LIN {X 0,Y 161.529,Z 676.326,A -85,B 0,C 180,E1 -24059.519,E2 -24059.519} C_VEL
LIN {X 0,Y 165.544,Z 667.107,A -85,B 0,C 180,E1 -24062.772,E2 -24062.772} C_VEL
LIN {X 0,Y 169.219,Z 658.14,A -85,B 0,C 180,E1 -24065.188,E2 -24065.188} C_VEL
LIN {X 0,Y 173.135,Z 647.011,A -85,B 0,C 180,E1 -24067.51,E2 -24067.51} C_VEL
LIN {X 0,Y 176.331,Z 636.142,A -85,B 0,C 180,E1 -24069.252,E2 -24069.252} C_VEL
LIN {X 0,Y 179.205,Z 624.067,A -85,B 0,C 180,E1 -24070.693,E2 -24070.693} C_VEL
LIN {X 0,Y 181.524,Z 611.447,A -85,B 0,C 180,E1 -24071.717,E2 -24071.717} C_VEL
LIN {X 0,Y 182.999,Z 598.442,A -85,B 0,C 180,E1 -24072.415,E2 -24072.415} C_VEL
LIN {X 0,Y 186.753,Z 537.772,A -85,B 0,C 180,E1 -24074.52,E2 -24074.52} C_VEL
LIN {X 0,Y 184.855,Z 513.189,A -85,B 0,C 180,E1 -24076.442,E2 -24076.442} C_VEL
LIN {X 0,Y 184.034,Z 505.216,A -85,B 0,C 180,E1 -24077.157,E2 -24077.157} C_VEL
LIN {X 0,Y 178.957,Z 494.02,A -85,B 0,C 180,E1 -24079.61,E2 -24079.61} C_VEL
LIN {X 0,Y 175.969,Z 487.994,A -85,B 0,C 180,E1 -24081.204,E2 -24081.204} C_VEL
LIN {X 0,Y 173.975,Z 480.034,A -85,B 0,C 180,E1 -24084.963,E2 -24084.963} C_VEL
LIN {X 0,Y 171.968,Z 473.299,A -85,B 0,C 180,E1 -24088.65,E2 -24088.65} C_VEL
LIN {X 0,Y 170.279,Z 468.344,A -85,B 0,C 180,E1 -24091.753,E2 -24091.753} C_VEL
LIN {X 0,Y 168.498,Z 463.406,A -85,B 0,C 180,E1 -24095.348,E2 -24095.348} C_VEL
LIN {X 0,Y 166.157,Z 457.892,A -85,B 0,C 180,E1 -24100.222,E2 -24100.222} C_VEL
LIN {X 0,Y 164.346,Z 453.629,A -85,B 0,C 180,E1 -24105.133,E2 -24105.133} C_VEL
LIN {X 0,Y 162.902,Z 450.174,A -85,B 0,C 180,E1 -24110.063,E2 -24110.063} C_VEL
LIN {X 0,Y 162.272,Z 448.989,A -85,B 0,C 180,E1 -24112.534,E2 -24112.534} C_VEL
LIN {X 0,Y 161.619,Z 446.459,A -85,B 0,C 180,E1 -24120,E2 -24120} C_VEL
LIN {X 0,Y 161.5,Z 446.45,A -85,B 0,C 180,E1 -24122.494,E2 -24122.494} C_VEL
LIN {X 0,Y 161.702,Z 447.367,A -85,B 0,C 180,E1 -24127.492,E2 -24127.492} C_VEL
LIN {X 0,Y 163.472,Z 450.303,A -85,B 0,C 180,E1 -24134.949,E2 -24134.949} C_VEL
LIN {X 0,Y 165.408,Z 453.727,A -85,B 0,C 180,E1 -24139.871,E2 -24139.871} C_VEL
LIN {X 0,Y 166.678,Z 455.735,A -85,B 0,C 180,E1 -24142.302,E2 -24142.302} C_VEL
LIN {X 0,Y 169.717,Z 461.04,A -85,B 0,C 180,E1 -24147.098,E2 -24147.098} C_VEL
LIN {X 0,Y 173.439,Z 467.697,A -85,B 0,C 180,E1 -24151.788,E2 -24151.788} C_VEL
LIN {X 0,Y 177.578,Z 476.226,A -85,B 0,C 180,E1 -24156.417,E2 -24156.417} C_VEL
LIN {X 0,Y 181.019,Z 483.948,A -85,B 0,C 180,E1 -24159.837,E2 -24159.837} C_VEL
LIN {X 0,Y 182.413,Z 487.889,A -85,B 0,C 180,E1 -24161.358,E2 -24161.358} C_VEL
LIN {X 0,Y 183.658,Z 492.595,A -85,B 0,C 180,E1 -24162.176,E2 -24162.176} C_VEL
LIN {X 0,Y 185.304,Z 519.809,A -85,B 0,C 180,E1 -24164.238,E2 -24164.238} C_VEL
LIN {X 0,Y 186.184,Z 541.587,A -85,B 0,C 180,E1 -24165.678,E2 -24165.678} C_VEL
LIN {X 0,Y 182.28,Z 603.538,A -85,B 0,C 180,E1 -24167.839,E2 -24167.839} C_VEL
LIN {X 0,Y 180.62,Z 616.473,A -85,B 0,C 180,E1 -24168.587,E2 -24168.587} C_VEL
LIN {X 0,Y 179.337,Z 623.194,A -85,B 0,C 180,E1 -24169.12,E2 -24169.12} C_VEL
LIN {X 0,Y 177.628,Z 628.814,A -85,B 0,C 180,E1 -24169.52,E2 -24169.52} C_VEL
LIN {X 0,Y 173.272,Z 637.686,A -85,B 0,C 180,E1 -24170.001,E2 -24170.001} C_VEL
LIN {X 0,Y 168.616,Z 646.095,A -85,B 0,C 180,E1 -24170.681,E2 -24170.681} C_VEL
LIN {X 0,Y 166.453,Z 651.018,A -85,B 0,C 180,E1 -24171.432,E2 -24171.432} C_VEL
LIN {X 0,Y 162.264,Z 661.871,A -85,B 0,C 180,E1 -24173.833,E2 -24173.833} C_VEL
LIN {X 0,Y 157.702,Z 672.349,A -85,B 0,C 180,E1 -24176.912,E2 -24176.912} C_VEL
LIN {X 0,Y 154.026,Z 680.047,A -85,B 0,C 180,E1 -24179.873,E2 -24179.873} C_VEL
LIN {X 0,Y 150.219,Z 687.553,A -85,B 0,C 180,E1 -24183.611,E2 -24183.611} C_VEL
LIN {X 0,Y 146.955,Z 693.583,A -85,B 0,C 180,E1 -24187.505,E2 -24187.505} C_VEL
LIN {X 0,Y 144.297,Z 698.343,A -85,B 0,C 180,E1 -24191.543,E2 -24191.543} C_VEL
LIN {X 0,Y 142.495,Z 701.977,A -85,B 0,C 180,E1 -24195.723,E2 -24195.723} C_VEL
LIN {X 0,Y 141.608,Z 703.849,A -85,B 0,C 180,E1 -24198.549,E2 -24198.549} C_VEL
LIN {X 0,Y 141.003,Z 705.258,A -85,B 0,C 180,E1 -24201.4,E2 -24201.4} C_VEL
LIN {X 0,Y 140.695,Z 706.254,A -85,B 0,C 180,E1 -24204.266,E2 -24204.266} C_VEL
LIN {X 0,Y 140.569,Z 707.048,A -85,B 0,C 180,E1 -24209.356,E2 -24209.356} C_VEL
LIN {X 0,Y 140.551,Z 706.847,A -85,B 0,C 180,E1 -24212.866,E2 -24212.866} C_VEL
LIN {X 0,Y 140.695,Z 706.23,A -85,B 0,C 180,E1 -24215.733,E2 -24215.733} C_VEL
LIN {X 0,Y 141.003,Z 705.224,A -85,B 0,C 180,E1 -24218.599,E2 -24218.599} C_VEL
LIN {X 0,Y 141.609,Z 703.795,A -85,B 0,C 180,E1 -24221.45,E2 -24221.45} C_VEL
LIN {X 0,Y 143.026,Z 700.831,A -85,B 0,C 180,E1 -24225.679,E2 -24225.679} C_VEL
LIN {X 0,Y 145.08,Z 696.809,A -85,B 0,C 180,E1 -24229.821,E2 -24229.821} C_VEL
LIN {X 0,Y 148.537,Z 690.612,A -85,B 0,C 180,E1 -24234.456,E2 -24234.456} C_VEL
LIN {X 0,Y 152.052,Z 684.024,A -85,B 0,C 180,E1 -24238.172,E2 -24238.172} C_VEL
LIN {X 0,Y 155.429,Z 676.931,A -85,B 0,C 180,E1 -24241.332,E2 -24241.332} C_VEL
LIN {X 0,Y 159.305,Z 668.576,A -85,B 0,C 180,E1 -24244.228,E2 -24244.228} C_VEL
LIN {X 0,Y 163.571,Z 658.245,A -85,B 0,C 180,E1 -24246.979,E2 -24246.979} C_VEL
LIN {X 0,Y 167.746,Z 646.617,A -85,B 0,C 180,E1 -24249.322,E2 -24249.322} C_VEL
LIN {X 0,Y 169.092,Z 643.157,A -85,B 0,C 180,E1 -24249.913,E2 -24249.913} C_VEL
LIN {X 0,Y 176.202,Z 640.592,A -85,B 0,C 180,E1 -24252.692,E2 -24252.692} C_VEL
LIN {X 0,Y 186.438,Z 636.605,A -85,B 0,C 180,E1 -24255.744,E2 -24255.744} C_VEL
LIN {X 0,Y 197.602,Z 631.417,A -85,B 0,C 180,E1 -24258.322,E2 -24258.322} C_VEL
LIN {X 0,Y 199.719,Z 630.307,A -85,B 0,C 180,E1 -24258.745,E2 -24258.745} C_VEL
LIN {X 0,Y 200.899,Z 629.352,A -85,B 0,C 180,E1 -24259.557,E2 -24259.557} C_VEL
LIN {X 0,Y 192.906,Z 631.179,A -85,B 0,C 180,E1 -24261.731,E2 -24261.731} C_VEL
LIN {X 0,Y 183.116,Z 632.283,A -85,B 0,C 180,E1 -24264.851,E2 -24264.851} C_VEL
LIN {X 0,Y 174.085,Z 632.009,A -85,B 0,C 180,E1 -24268.344,E2 -24268.344} C_VEL
LIN {X 0,Y 166.006,Z 630.276,A -85,B 0,C 180,E1 -24272.245,E2 -24272.245} C_VEL
LIN {X 0,Y 158.996,Z 627.135,A -85,B 0,C 180,E1 -24276.558,E2 -24276.558} C_VEL
LIN {X 0,Y 153.197,Z 622.556,A -85,B 0,C 180,E1 -24281.269,E2 -24281.269} C_VEL
LIN {X 0,Y 148.739,Z 616.364,A -85,B 0,C 180,E1 -24286.335,E2 -24286.335} C_VEL
LIN {X 0,Y 146.114,Z 609.561,A -85,B 0,C 180,E1 -24291.007,E2 -24291.007} C_VEL
LIN {X 0,Y 144.181,Z 601.237,A -85,B 0,C 180,E1 -24295.807,E2 -24295.807} C_VEL
LIN {X 0,Y 143.45,Z 590.998,A -85,B 0,C 180,E1 -24300.702,E2 -24300.702} C_VEL
LIN {X 0,Y 143.461,Z 580.348,A -85,B 0,C 180,E1 -24304.918,E2 -24304.918} C_VEL
LIN {X 0,Y 143.996,Z 568.578,A -85,B 0,C 180,E1 -24308.773,E2 -24308.773} C_VEL
LIN {X 0,Y 144.72,Z 555.919,A -85,B 0,C 180,E1 -24312.081,E2 -24312.081} C_VEL
LIN {X 0,Y 145.46,Z 543.621,A -85,B 0,C 180,E1 -24314.694,E2 -24314.694} C_VEL
LIN {X 0,Y 146.296,Z 529.161,A -85,B 0,C 180,E1 -24317.112,E2 -24317.112} C_VEL
LIN {X 0,Y 146.975,Z 515.38,A -85,B 0,C 180,E1 -24318.831,E2 -24318.831} C_VEL
LIN {X 0,Y 147.665,Z 492.766,A -85,B 0,C 180,E1 -24321.096,E2 -24321.096} C_VEL
LIN {X 0,Y 147.855,Z 488.31,A -85,B 0,C 180,E1 -24321.891,E2 -24321.891} C_VEL
LIN {X 0,Y 148.091,Z 487.68,A -85,B 0,C 180,E1 -24322.313,E2 -24322.313} C_VEL
LIN {X 0,Y 149.825,Z 486.897,A -85,B 0,C 180,E1 -24323.498,E2 -24323.498} C_VEL
LIN {X 0,Y 152.829,Z 484.252,A -85,B 0,C 180,E1 -24324.449,E2 -24324.449} C_VEL
LIN {X 0,Y 154.839,Z 483.406,A -85,B 0,C 180,E1 -24325.545,E2 -24325.545} C_VEL
LIN {X 0,Y 160.173,Z 479.672,A -85,B 0,C 180,E1 -24327.434,E2 -24327.434} C_VEL
LIN {X 0,Y 162.59,Z 478.361,A -85,B 0,C 180,E1 -24328.391,E2 -24328.391} C_VEL
LIN {X 0,Y 165.368,Z 476.481,A -85,B 0,C 180,E1 -24329.258,E2 -24329.258} C_VEL
LIN {X 0,Y 166.775,Z 477.154,A -85,B 0,C 180,E1 -24330.377,E2 -24330.377} C_VEL
LIN {X 0,Y 168.809,Z 483.952,A -85,B 0,C 180,E1 -24334.196,E2 -24334.196} C_VEL
LIN {X 0,Y 169.895,Z 488.503,A -85,B 0,C 180,E1 -24336.503,E2 -24336.503} C_VEL
LIN {X 0,Y 174.656,Z 497.876,A -85,B 0,C 180,E1 -24339.176,E2 -24339.176} C_VEL
LIN {X 0,Y 178.713,Z 507.05,A -85,B 0,C 180,E1 -24341.295,E2 -24341.295} C_VEL
LIN {X 0,Y 179.393,Z 509.152,A -85,B 0,C 180,E1 -24341.666,E2 -24341.666} C_VEL
LIN {X 0,Y 181.143,Z 532.748,A -85,B 0,C 180,E1 -24343.63,E2 -24343.63} C_VEL
LIN {X 0,Y 181.538,Z 539.6,A -85,B 0,C 180,E1 -24344.143,E2 -24344.143} C_VEL
LIN {X 0,Y 177.35,Z 602.381,A -85,B 0,C 180,E1 -24346.383,E2 -24346.383} C_VEL
LIN {X 0,Y 175.415,Z 615.477,A -85,B 0,C 180,E1 -24347.168,E2 -24347.168} C_VEL
LIN {X 0,Y 172.761,Z 628.498,A -85,B 0,C 180,E1 -24348.425,E2 -24348.425} C_VEL
LIN {X 0,Y 169.587,Z 640.39,A -85,B 0,C 180,E1 -24350.033,E2 -24350.033} C_VEL
LIN {X 0,Y 165.778,Z 651.672,A -85,B 0,C 180,E1 -24352.069,E2 -24352.069} C_VEL
LIN {X 0,Y 161.788,Z 661.855,A -85,B 0,C 180,E1 -24354.479,E2 -24354.479} C_VEL
LIN {X 0,Y 158.169,Z 670.201,A -85,B 0,C 180,E1 -24357.023,E2 -24357.023} C_VEL
LIN {X 0,Y 154.607,Z 677.898,A -85,B 0,C 180,E1 -24359.998,E2 -24359.998} C_VEL
LIN {X 0,Y 150.701,Z 685.393,A -85,B 0,C 180,E1 -24363.702,E2 -24363.702} C_VEL
LIN {X 0,Y 147.336,Z 691.406,A -85,B 0,C 180,E1 -24367.567,E2 -24367.567} C_VEL
LIN {X 0,Y 144.701,Z 696.159,A -85,B 0,C 180,E1 -24371.597,E2 -24371.597} C_VEL
LIN {X 0,Y 142.761,Z 699.794,A -85,B 0,C 180,E1 -24375.751,E2 -24375.751} C_VEL
LIN {X 0,Y 141.822,Z 701.664,A -85,B 0,C 180,E1 -24378.567,E2 -24378.567} C_VEL
LIN {X 0,Y 141.13,Z 703.088,A -85,B 0,C 180,E1 -24381.409,E2 -24381.409} C_VEL
LIN {X 0,Y 140.727,Z 704.087,A -85,B 0,C 180,E1 -24384.268,E2 -24384.268} C_VEL
LIN {X 0,Y 140.538,Z 704.701,A -85,B 0,C 180,E1 -24387.134,E2 -24387.134} C_VEL
LIN {X 0,Y 140.528,Z 704.932,A -85,B 0,C 180,E1 -24390,E2 -24390} C_VEL
LIN {X 0,Y 140.538,Z 704.731,A -85,B 0,C 180,E1 -24392.867,E2 -24392.867} C_VEL
LIN {X 0,Y 140.71,Z 704.137,A -85,B 0,C 180,E1 -24395.733,E2 -24395.733} C_VEL
LIN {X 0,Y 141.083,Z 703.158,A -85,B 0,C 180,E1 -24398.595,E2 -24398.595} C_VEL
LIN {X 0,Y 141.74,Z 701.773,A -85,B 0,C 180,E1 -24401.44,E2 -24401.44} C_VEL
LIN {X 0,Y 143.28,Z 698.869,A -85,B 0,C 180,E1 -24405.652,E2 -24405.652} C_VEL
LIN {X 0,Y 145.379,Z 694.923,A -85,B 0,C 180,E1 -24409.78,E2 -24409.78} C_VEL
LIN {X 0,Y 148.322,Z 689.807,A -85,B 0,C 180,E1 -24413.751,E2 -24413.751} C_VEL
LIN {X 0,Y 151.813,Z 683.36,A -85,B 0,C 180,E1 -24417.577,E2 -24417.577} C_VEL
LIN {X 0,Y 155.861,Z 675.352,A -85,B 0,C 180,E1 -24421.234,E2 -24421.234} C_VEL
LIN {X 0,Y 159.596,Z 667.153,A -85,B 0,C 180,E1 -24424.158,E2 -24424.158} C_VEL
LIN {X 0,Y 163.938,Z 657.038,A -85,B 0,C 180,E1 -24426.883,E2 -24426.883} C_VEL
LIN {X 0,Y 168.049,Z 645.661,A -85,B 0,C 180,E1 -24429.239,E2 -24429.239} C_VEL
LIN {X 0,Y 171.384,Z 634.406,A -85,B 0,C 180,E1 -24431.005,E2 -24431.005} C_VEL
LIN {X 0,Y 174.427,Z 621.607,A -85,B 0,C 180,E1 -24432.446,E2 -24432.446} C_VEL
LIN {X 0,Y 176.664,Z 609.011,A -85,B 0,C 180,E1 -24433.416,E2 -24433.416} C_VEL
LIN {X 0,Y 178.074,Z 595.759,A -85,B 0,C 180,E1 -24434.041,E2 -24434.041} C_VEL
LIN {X 0,Y 181.707,Z 538.828,A -85,B 0,C 180,E1 -24436.043,E2 -24436.043} C_VEL
LIN {X 0,Y 180.027,Z 514.977,A -85,B 0,C 180,E1 -24437.973,E2 -24437.973} C_VEL
LIN {X 0,Y 179.352,Z 508.348,A -85,B 0,C 180,E1 -24438.604,E2 -24438.604} C_VEL
LIN {X 0,Y 174.464,Z 497.305,A -85,B 0,C 180,E1 -24441.159,E2 -24441.159} C_VEL
LIN {X 0,Y 169.725,Z 487.967,A -85,B 0,C 180,E1 -24443.908,E2 -24443.908} C_VEL
LIN {X 0,Y 167.852,Z 480.601,A -85,B 0,C 180,E1 -24447.79,E2 -24447.79} C_VEL
LIN {X 0,Y 166.296,Z 475.411,A -85,B 0,C 180,E1 -24450.921,E2 -24450.921} C_VEL
LIN {X 0,Y 164.426,Z 470.181,A -85,B 0,C 180,E1 -24454.695,E2 -24454.695} C_VEL
LIN {X 0,Y 162.79,Z 465.679,A -85,B 0,C 180,E1 -24458.471,E2 -24458.471} C_VEL
LIN {X 0,Y 161.257,Z 461.982,A -85,B 0,C 180,E1 -24462.237,E2 -24462.237} C_VEL
LIN {X 0,Y 159.754,Z 458.091,A -85,B 0,C 180,E1 -24467.293,E2 -24467.293} C_VEL
LIN {X 0,Y 159.225,Z 456.473,A -85,B 0,C 180,E1 -24469.831,E2 -24469.831} C_VEL
LIN {X 0,Y 158.634,Z 455.181,A -85,B 0,C 180,E1 -24472.362,E2 -24472.362} C_VEL
LIN {X 0,Y 157.973,Z 452.588,A -85,B 0,C 180,E1 -24480,E2 -24480} C_VEL
LIN {X 0,Y 157.969,Z 452.641,A -85,B 0,C 180,E1 -24482.55,E2 -24482.55} C_VEL
LIN {X 0,Y 158.328,Z 453.67,A -85,B 0,C 180,E1 -24487.653,E2 -24487.653} C_VEL
LIN {X 0,Y 160.107,Z 456.758,A -85,B 0,C 180,E1 -24495.27,E2 -24495.27} C_VEL
LIN {X 0,Y 162.611,Z 461.061,A -85,B 0,C 180,E1 -24501.312,E2 -24501.312} C_VEL
LIN {X 0,Y 165.743,Z 466.703,A -85,B 0,C 180,E1 -24506.574,E2 -24506.574} C_VEL
LIN {X 0,Y 168.843,Z 472.526,A -85,B 0,C 180,E1 -24510.816,E2 -24510.816} C_VEL
LIN {X 0,Y 172.221,Z 479.503,A -85,B 0,C 180,E1 -24514.842,E2 -24514.842} C_VEL
LIN {X 0,Y 175.924,Z 488.125,A -85,B 0,C 180,E1 -24518.953,E2 -24518.953} C_VEL
LIN {X 0,Y 178.149,Z 492.16,A -85,B 0,C 180,E1 -24520.148,E2 -24520.148} C_VEL
LIN {X 0,Y 178.999,Z 495.228,A -85,B 0,C 180,E1 -24520.656,E2 -24520.656} C_VEL
LIN {X 0,Y 180.507,Z 523.357,A -85,B 0,C 180,E1 -24522.85,E2 -24522.85} C_VEL
LIN {X 0,Y 181.158,Z 542.035,A -85,B 0,C 180,E1 -24524.124,E2 -24524.124} C_VEL
LIN {X 0,Y 177.056,Z 603.874,A -85,B 0,C 180,E1 -24526.309,E2 -24526.309} C_VEL
LIN {X 0,Y 175.358,Z 616.466,A -85,B 0,C 180,E1 -24527.052,E2 -24527.052} C_VEL
LIN {X 0,Y 172.683,Z 629.321,A -85,B 0,C 180,E1 -24528.206,E2 -24528.206} C_VEL
LIN {X 0,Y 169.696,Z 640.745,A -85,B 0,C 180,E1 -24529.675,E2 -24529.675} C_VEL
LIN {X 0,Y 166.453,Z 651.018,A -85,B 0,C 180,E1 -24531.432,E2 -24531.432} C_VEL
LIN {X 0,Y 164.182,Z 655.911,A -85,B 0,C 180,E1 -24532.271,E2 -24532.271} C_VEL
LIN {X 0,Y 158.789,Z 663.497,A -85,B 0,C 180,E1 -24533.492,E2 -24533.492} C_VEL
LIN {X 0,Y 153.178,Z 670.57,A -85,B 0,C 180,E1 -24535.004,E2 -24535.004} C_VEL
LIN {X 0,Y 150.621,Z 674.63,A -85,B 0,C 180,E1 -24536.298,E2 -24536.298} C_VEL
LIN {X 0,Y 146.746,Z 682.242,A -85,B 0,C 180,E1 -24539.549,E2 -24539.549} C_VEL
LIN {X 0,Y 143.238,Z 688.611,A -85,B 0,C 180,E1 -24543.008,E2 -24543.008} C_VEL
LIN {X 0,Y 140.417,Z 693.532,A -85,B 0,C 180,E1 -24546.396,E2 -24546.396} C_VEL
LIN {X 0,Y 137.559,Z 698.291,A -85,B 0,C 180,E1 -24550.604,E2 -24550.604} C_VEL
LIN {X 0,Y 135.585,Z 701.924,A -85,B 0,C 180,E1 -24554.979,E2 -24554.979} C_VEL
LIN {X 0,Y 134.626,Z 703.796,A -85,B 0,C 180,E1 -24557.947,E2 -24557.947} C_VEL
LIN {X 0,Y 133.976,Z 705.205,A -85,B 0,C 180,E1 -24560.945,E2 -24560.945} C_VEL
LIN {X 0,Y 133.631,Z 706.201,A -85,B 0,C 180,E1 -24563.962,E2 -24563.962} C_VEL
LIN {X 0,Y 133.471,Z 706.808,A -85,B 0,C 180,E1 -24566.981,E2 -24566.981} C_VEL
LIN {X 0,Y 133.499,Z 707.02,A -85,B 0,C 180,E1 -24570,E2 -24570} C_VEL
LIN {X 0,Y 133.47,Z 706.793,A -85,B 0,C 180,E1 -24573.018,E2 -24573.018} C_VEL
LIN {X 0,Y 133.63,Z 706.175,A -85,B 0,C 180,E1 -24576.037,E2 -24576.037} C_VEL
LIN {X 0,Y 133.976,Z 705.169,A -85,B 0,C 180,E1 -24579.054,E2 -24579.054} C_VEL
LIN {X 0,Y 134.627,Z 703.74,A -85,B 0,C 180,E1 -24582.052,E2 -24582.052} C_VEL
LIN {X 0,Y 136.174,Z 700.776,A -85,B 0,C 180,E1 -24586.49,E2 -24586.49} C_VEL
LIN {X 0,Y 138.412,Z 696.755,A -85,B 0,C 180,E1 -24590.82,E2 -24590.82} C_VEL
LIN {X 0,Y 142.07,Z 690.558,A -85,B 0,C 180,E1 -24595.648,E2 -24595.648} C_VEL
LIN {X 0,Y 146.049,Z 683.455,A -85,B 0,C 180,E1 -24599.776,E2 -24599.776} C_VEL
LIN {X 0,Y 150.164,Z 675.323,A -85,B 0,C 180,E1 -24603.362,E2 -24603.362} C_VEL
LIN {X 0,Y 154.361,Z 666.605,A -85,B 0,C 180,E1 -24606.291,E2 -24606.291} C_VEL
LIN {X 0,Y 158.907,Z 655.881,A -85,B 0,C 180,E1 -24609.067,E2 -24609.067} C_VEL
LIN {X 0,Y 162.858,Z 645.067,A -85,B 0,C 180,E1 -24611.155,E2 -24611.155} C_VEL
LIN {X 0,Y 164.166,Z 642.142,A -85,B 0,C 180,E1 -24611.674,E2 -24611.674} C_VEL
LIN {X 0,Y 171.063,Z 640.15,A -85,B 0,C 180,E1 -24614.301,E2 -24614.301} C_VEL
LIN {X 0,Y 181.547,Z 636.713,A -85,B 0,C 180,E1 -24617.351,E2 -24617.351} C_VEL
LIN {X 0,Y 190.232,Z 633.287,A -85,B 0,C 180,E1 -24619.357,E2 -24619.357} C_VEL
LIN {X 0,Y 189.199,Z 633.24,A -85,B 0,C 180,E1 -24620.008,E2 -24620.008} C_VEL
LIN {X 0,Y 182.475,Z 633.879,A -85,B 0,C 180,E1 -24621.958,E2 -24621.958} C_VEL
LIN {X 0,Y 172.7,Z 633.752,A -85,B 0,C 180,E1 -24625.269,E2 -24625.269} C_VEL
LIN {X 0,Y 163.858,Z 632.238,A -85,B 0,C 180,E1 -24629.023,E2 -24629.023} C_VEL
LIN {X 0,Y 156,Z 629.292,A -85,B 0,C 180,E1 -24633.223,E2 -24633.223} C_VEL
LIN {X 0,Y 149.33,Z 624.929,A -85,B 0,C 180,E1 -24637.882,E2 -24637.882} C_VEL
LIN {X 0,Y 143.999,Z 619.088,A -85,B 0,C 180,E1 -24642.972,E2 -24642.972} C_VEL
LIN {X 0,Y 140.286,Z 611.576,A -85,B 0,C 180,E1 -24648.44,E2 -24648.44} C_VEL
LIN {X 0,Y 137.94,Z 603.393,A -85,B 0,C 180,E1 -24653.417,E2 -24653.417} C_VEL
LIN {X 0,Y 136.694,Z 593.477,A -85,B 0,C 180,E1 -24658.527,E2 -24658.527} C_VEL
LIN {X 0,Y 136.479,Z 583.189,A -85,B 0,C 180,E1 -24662.952,E2 -24662.952} C_VEL
LIN {X 0,Y 136.852,Z 571.757,A -85,B 0,C 180,E1 -24667.006,E2 -24667.006} C_VEL
LIN {X 0,Y 137.419,Z 560.623,A -85,B 0,C 180,E1 -24670.312,E2 -24670.312} C_VEL
LIN {X 0,Y 138.073,Z 549.186,A -85,B 0,C 180,E1 -24673.08,E2 -24673.08} C_VEL
LIN {X 0,Y 138.971,Z 533.049,A -85,B 0,C 180,E1 -24676.176,E2 -24676.176} C_VEL
LIN {X 0,Y 139.44,Z 524.996,A -85,B 0,C 180,E1 -24677.792,E2 -24677.792} C_VEL
LIN {X 0,Y 139.758,Z 522.696,A -85,B 0,C 180,E1 -24678.603,E2 -24678.603} C_VEL
LIN {X 0,Y 140.364,Z 521.75,A -85,B 0,C 180,E1 -24679.373,E2 -24679.373} C_VEL
LIN {X 0,Y 141.679,Z 518.777,A -85,B 0,C 180,E1 -24680.413,E2 -24680.413} C_VEL
LIN {X 0,Y 143.518,Z 513.065,A -85,B 0,C 180,E1 -24681.549,E2 -24681.549} C_VEL
LIN {X 0,Y 147.072,Z 499.47,A -85,B 0,C 180,E1 -24683.219,E2 -24683.219} C_VEL
LIN {X 0,Y 148.576,Z 493.924,A -85,B 0,C 180,E1 -24683.893,E2 -24683.893} C_VEL
LIN {X 0,Y 150.073,Z 492.752,A -85,B 0,C 180,E1 -24685.02,E2 -24685.02} C_VEL
LIN {X 0,Y 152.013,Z 489.85,A -85,B 0,C 180,E1 -24686.238,E2 -24686.238} C_VEL
LIN {X 0,Y 153.569,Z 488.674,A -85,B 0,C 180,E1 -24687.235,E2 -24687.235} C_VEL
LIN {X 0,Y 158.932,Z 484.913,A -85,B 0,C 180,E1 -24689.106,E2 -24689.106} C_VEL
LIN {X 0,Y 161.439,Z 483.58,A -85,B 0,C 180,E1 -24690.042,E2 -24690.042} C_VEL
LIN {X 0,Y 162.751,Z 484.509,A -85,B 0,C 180,E1 -24691.211,E2 -24691.211} C_VEL
LIN {X 0,Y 163.667,Z 488.248,A -85,B 0,C 180,E1 -24693.403,E2 -24693.403} C_VEL
LIN {X 0,Y 167.785,Z 496.259,A -85,B 0,C 180,E1 -24696.091,E2 -24696.091} C_VEL
LIN {X 0,Y 171.493,Z 503.922,A -85,B 0,C 180,E1 -24698.265,E2 -24698.265} C_VEL
LIN {X 0,Y 174.778,Z 511.715,A -85,B 0,C 180,E1 -24700.099,E2 -24700.099} C_VEL
LIN {X 0,Y 176.255,Z 533.448,A -85,B 0,C 180,E1 -24701.98,E2 -24701.98} C_VEL
LIN {X 0,Y 176.616,Z 539.816,A -85,B 0,C 180,E1 -24702.488,E2 -24702.488} C_VEL
LIN {X 0,Y 172.26,Z 602.734,A -85,B 0,C 180,E1 -24704.775,E2 -24704.775} C_VEL
LIN {X 0,Y 170.296,Z 615.503,A -85,B 0,C 180,E1 -24705.55,E2 -24705.55} C_VEL
LIN {X 0,Y 167.521,Z 628.535,A -85,B 0,C 180,E1 -24706.815,E2 -24706.815} C_VEL
LIN {X 0,Y 164.215,Z 640.434,A -85,B 0,C 180,E1 -24708.443,E2 -24708.443} C_VEL
LIN {X 0,Y 160.249,Z 651.719,A -85,B 0,C 180,E1 -24710.512,E2 -24710.512} C_VEL
LIN {X 0,Y 156.073,Z 661.904,A -85,B 0,C 180,E1 -24712.967,E2 -24712.967} C_VEL
LIN {X 0,Y 152.238,Z 670.253,A -85,B 0,C 180,E1 -24715.562,E2 -24715.562} C_VEL
LIN {X 0,Y 147.773,Z 679.293,A -85,B 0,C 180,E1 -24719.252,E2 -24719.252} C_VEL
LIN {X 0,Y 143.745,Z 686.544,A -85,B 0,C 180,E1 -24723.112,E2 -24723.112} C_VEL
LIN {X 0,Y 139.751,Z 693.19,A -85,B 0,C 180,E1 -24727.842,E2 -24727.842} C_VEL
LIN {X 0,Y 137.215,Z 697.553,A -85,B 0,C 180,E1 -24732.103,E2 -24732.103} C_VEL
LIN {X 0,Y 135.874,Z 699.848,A -85,B 0,C 180,E1 -24735.012,E2 -24735.012} C_VEL
LIN {X 0,Y 134.85,Z 701.719,A -85,B 0,C 180,E1 -24737.968,E2 -24737.968} C_VEL
LIN {X 0,Y 134.108,Z 703.143,A -85,B 0,C 180,E1 -24740.955,E2 -24740.955} C_VEL
LIN {X 0,Y 133.466,Z 704.755,A -85,B 0,C 180,E1 -24746.982,E2 -24746.982} C_VEL
LIN {X 0,Y 133.45,Z 704.986,A -85,B 0,C 180,E1 -24750,E2 -24750} C_VEL
LIN {X 0,Y 133.465,Z 704.785,A -85,B 0,C 180,E1 -24753.019,E2 -24753.019} C_VEL
LIN {X 0,Y 133.645,Z 704.19,A -85,B 0,C 180,E1 -24756.038,E2 -24756.038} C_VEL
LIN {X 0,Y 134.068,Z 703.211,A -85,B 0,C 180,E1 -24759.049,E2 -24759.049} C_VEL
LIN {X 0,Y 134.779,Z 701.826,A -85,B 0,C 180,E1 -24762.04,E2 -24762.04} C_VEL
LIN {X 0,Y 136.437,Z 698.922,A -85,B 0,C 180,E1 -24766.458,E2 -24766.458} C_VEL
LIN {X 0,Y 138.697,Z 694.975,A -85,B 0,C 180,E1 -24770.776,E2 -24770.776} C_VEL
LIN {X 0,Y 141.843,Z 689.857,A -85,B 0,C 180,E1 -24774.908,E2 -24774.908} C_VEL
LIN {X 0,Y 145.552,Z 683.41,A -85,B 0,C 180,E1 -24778.873,E2 -24778.873} C_VEL
LIN {X 0,Y 149.672,Z 675.688,A -85,B 0,C 180,E1 -24782.524,E2 -24782.524} C_VEL
LIN {X 0,Y 153.77,Z 667.198,A -85,B 0,C 180,E1 -24785.644,E2 -24785.644} C_VEL
LIN {X 0,Y 157.819,Z 658.223,A -85,B 0,C 180,E1 -24788.162,E2 -24788.162} C_VEL
LIN {X 0,Y 162.114,Z 647.086,A -85,B 0,C 180,E1 -24790.564,E2 -24790.564} C_VEL
LIN {X 0,Y 165.596,Z 636.203,A -85,B 0,C 180,E1 -24792.358,E2 -24792.358} C_VEL
LIN {X 0,Y 168.71,Z 624.102,A -85,B 0,C 180,E1 -24793.833,E2 -24793.833} C_VEL
LIN {X 0,Y 171.303,Z 610.821,A -85,B 0,C 180,E1 -24794.918,E2 -24794.918} C_VEL
LIN {X 0,Y 172.837,Z 597.976,A -85,B 0,C 180,E1 -24795.601,E2 -24795.601} C_VEL
LIN {X 0,Y 176.792,Z 539.57,A -85,B 0,C 180,E1 -24797.671,E2 -24797.671} C_VEL
LIN {X 0,Y 175.298,Z 516.482,A -85,B 0,C 180,E1 -24799.619,E2 -24799.619} C_VEL
LIN {X 0,Y 174.885,Z 511.695,A -85,B 0,C 180,E1 -24800.077,E2 -24800.077} C_VEL
LIN {X 0,Y 170.468,Z 501.504,A -85,B 0,C 180,E1 -24802.567,E2 -24802.567} C_VEL
LIN {X 0,Y 165.419,Z 491.576,A -85,B 0,C 180,E1 -24805.648,E2 -24805.648} C_VEL
LIN {X 0,Y 163.562,Z 487.994,A -85,B 0,C 180,E1 -24806.964,E2 -24806.964} C_VEL
LIN {X 0,Y 161.951,Z 481.711,A -85,B 0,C 180,E1 -24810.721,E2 -24810.721} C_VEL
LIN {X 0,Y 160.456,Z 476.936,A -85,B 0,C 180,E1 -24814.023,E2 -24814.023} C_VEL
LIN {X 0,Y 158.541,Z 471.503,A -85,B 0,C 180,E1 -24818.579,E2 -24818.579} C_VEL
LIN {X 0,Y 156.912,Z 467.237,A -85,B 0,C 180,E1 -24823.074,E2 -24823.074} C_VEL
LIN {X 0,Y 155.838,Z 464.31,A -85,B 0,C 180,E1 -24826.968,E2 -24826.968} C_VEL
LIN {X 0,Y 155.337,Z 462.656,A -85,B 0,C 180,E1 -24829.573,E2 -24829.573} C_VEL
LIN {X 0,Y 154.927,Z 461.365,A -85,B 0,C 180,E1 -24832.178,E2 -24832.178} C_VEL
LIN {X 0,Y 154.342,Z 458.712,A -85,B 0,C 180,E1 -24840,E2 -24840} C_VEL
LIN {X 0,Y 154.348,Z 458.755,A -85,B 0,C 180,E1 -24842.61,E2 -24842.61} C_VEL
LIN {X 0,Y 154.722,Z 459.874,A -85,B 0,C 180,E1 -24847.832,E2 -24847.832} C_VEL
LIN {X 0,Y 155.857,Z 461.88,A -85,B 0,C 180,E1 -24853.03,E2 -24853.03} C_VEL
LIN {X 0,Y 156.705,Z 463.223,A -85,B 0,C 180,E1 -24855.61,E2 -24855.61} C_VEL
LIN {X 0,Y 158.777,Z 466.836,A -85,B 0,C 180,E1 -24860.739,E2 -24860.739} C_VEL
LIN {X 0,Y 161.517,Z 472,A -85,B 0,C 180,E1 -24865.793,E2 -24865.793} C_VEL
LIN {X 0,Y 164.025,Z 476.963,A -85,B 0,C 180,E1 -24869.521,E2 -24869.521} C_VEL
LIN {X 0,Y 166.875,Z 482.794,A -85,B 0,C 180,E1 -24873.196,E2 -24873.196} C_VEL
LIN {X 0,Y 169.682,Z 489.044,A -85,B 0,C 180,E1 -24876.399,E2 -24876.399} C_VEL
LIN {X 0,Y 174.111,Z 496.368,A -85,B 0,C 180,E1 -24878.813,E2 -24878.813} C_VEL
LIN {X 0,Y 174.544,Z 498.475,A -85,B 0,C 180,E1 -24879.125,E2 -24879.125} C_VEL
LIN {X 0,Y 175.874,Z 529.031,A -85,B 0,C 180,E1 -24881.535,E2 -24881.535} C_VEL
LIN {X 0,Y 176.144,Z 544.225,A -85,B 0,C 180,E1 -24882.54,E2 -24882.54} C_VEL
LIN {X 0,Y 171.971,Z 604.227,A -85,B 0,C 180,E1 -24884.692,E2 -24884.692} C_VEL
LIN {X 0,Y 170.107,Z 617.193,A -85,B 0,C 180,E1 -24885.486,E2 -24885.486} C_VEL
LIN {X 0,Y 167.2,Z 630.397,A -85,B 0,C 180,E1 -24886.711,E2 -24886.711} C_VEL
LIN {X 0,Y 163.855,Z 642.358,A -85,B 0,C 180,E1 -24888.331,E2 -24888.331} C_VEL
LIN {X 0,Y 159.914,Z 653.706,A -85,B 0,C 180,E1 -24890.412,E2 -24890.412} C_VEL
LIN {X 0,Y 155.693,Z 663.938,A -85,B 0,C 180,E1 -24892.86,E2 -24892.86} C_VEL
LIN {X 0,Y 151.798,Z 672.303,A -85,B 0,C 180,E1 -24895.447,E2 -24895.447} C_VEL
LIN {X 0,Y 150.621,Z 674.63,A -85,B 0,C 180,E1 -24896.298,E2 -24896.298} C_VEL
LIN {X 0,Y 148.091,Z 678.526,A -85,B 0,C 180,E1 -24897.71,E2 -24897.71} C_VEL
LIN {X 0,Y 142.468,Z 684.42,A -85,B 0,C 180,E1 -24899.943,E2 -24899.943} C_VEL
LIN {X 0,Y 136.895,Z 689.698,A -85,B 0,C 180,E1 -24902.527,E2 -24902.527} C_VEL
LIN {X 0,Y 134.516,Z 692.558,A -85,B 0,C 180,E1 -24904.465,E2 -24904.465} C_VEL
LIN {X 0,Y 130.87,Z 698.239,A -85,B 0,C 180,E1 -24909.569,E2 -24909.569} C_VEL
LIN {X 0,Y 128.711,Z 701.871,A -85,B 0,C 180,E1 -24914.156,E2 -24914.156} C_VEL
LIN {X 0,Y 127.671,Z 703.743,A -85,B 0,C 180,E1 -24917.279,E2 -24917.279} C_VEL
LIN {X 0,Y 126.951,Z 705.151,A -85,B 0,C 180,E1 -24920.44,E2 -24920.44} C_VEL
LIN {X 0,Y 126.563,Z 706.147,A -85,B 0,C 180,E1 -24923.623,E2 -24923.623} C_VEL
LIN {X 0,Y 126.384,Z 706.754,A -85,B 0,C 180,E1 -24926.812,E2 -24926.812} C_VEL
LIN {X 0,Y 126.421,Z 706.966,A -85,B 0,C 180,E1 -24930,E2 -24930} C_VEL
LIN {X 0,Y 126.384,Z 706.739,A -85,B 0,C 180,E1 -24933.187,E2 -24933.187} C_VEL
LIN {X 0,Y 126.563,Z 706.121,A -85,B 0,C 180,E1 -24936.376,E2 -24936.376} C_VEL
LIN {X 0,Y 126.951,Z 705.115,A -85,B 0,C 180,E1 -24939.56,E2 -24939.56} C_VEL
LIN {X 0,Y 127.672,Z 703.685,A -85,B 0,C 180,E1 -24942.72,E2 -24942.72} C_VEL
LIN {X 0,Y 129.358,Z 700.722,A -85,B 0,C 180,E1 -24947.386,E2 -24947.386} C_VEL
LIN {X 0,Y 131.795,Z 696.701,A -85,B 0,C 180,E1 -24951.917,E2 -24951.917} C_VEL
LIN {X 0,Y 135.656,Z 690.504,A -85,B 0,C 180,E1 -24956.956,E2 -24956.956} C_VEL
LIN {X 0,Y 139.6,Z 683.93,A -85,B 0,C 180,E1 -24960.938,E2 -24960.938} C_VEL
LIN {X 0,Y 143.451,Z 676.827,A -85,B 0,C 180,E1 -24964.292,E2 -24964.292} C_VEL
LIN {X 0,Y 147.789,Z 668.475,A -85,B 0,C 180,E1 -24967.323,E2 -24967.323} C_VEL
LIN {X 0,Y 152.474,Z 658.148,A -85,B 0,C 180,E1 -24970.188,E2 -24970.188} C_VEL
LIN {X 0,Y 157.042,Z 646.528,A -85,B 0,C 180,E1 -24972.6,E2 -24972.6} C_VEL
LIN {X 0,Y 159.248,Z 641.163,A -85,B 0,C 180,E1 -24973.487,E2 -24973.487} C_VEL
LIN {X 0,Y 171.324,Z 638.165,A -85,B 0,C 180,E1 -24977.594,E2 -24977.594} C_VEL
LIN {X 0,Y 178.22,Z 636.155,A -85,B 0,C 180,E1 -24979.387,E2 -24979.387} C_VEL
LIN {X 0,Y 179.048,Z 635.647,A -85,B 0,C 180,E1 -24980,E2 -24980} C_VEL
LIN {X 0,Y 171.937,Z 635.493,A -85,B 0,C 180,E1 -24982.184,E2 -24982.184} C_VEL
LIN {X 0,Y 162.281,Z 634.127,A -85,B 0,C 180,E1 -24985.737,E2 -24985.737} C_VEL
LIN {X 0,Y 153.619,Z 631.395,A -85,B 0,C 180,E1 -24989.785,E2 -24989.785} C_VEL
LIN {X 0,Y 146.079,Z 627.233,A -85,B 0,C 180,E1 -24994.342,E2 -24994.342} C_VEL
LIN {X 0,Y 139.827,Z 621.623,A -85,B 0,C 180,E1 -24999.401,E2 -24999.401} C_VEL
LIN {X 0,Y 135.105,Z 614.454,A -85,B 0,C 180,E1 -25004.924,E2 -25004.924} C_VEL
LIN {X 0,Y 132.285,Z 606.703,A -85,B 0,C 180,E1 -25010.057,E2 -25010.057} C_VEL
LIN {X 0,Y 130.35,Z 597.252,A -85,B 0,C 180,E1 -25015.361,E2 -25015.361} C_VEL
LIN {X 0,Y 129.632,Z 585.825,A -85,B 0,C 180,E1 -25020.777,E2 -25020.777} C_VEL
LIN {X 0,Y 129.788,Z 574.838,A -85,B 0,C 180,E1 -25025.048,E2 -25025.048} C_VEL
LIN {X 0,Y 130.318,Z 561.439,A -85,B 0,C 180,E1 -25029.703,E2 -25029.703} C_VEL
LIN {X 0,Y 130.513,Z 558.546,A -85,B 0,C 180,E1 -25031.158,E2 -25031.158} C_VEL
LIN {X 0,Y 131.312,Z 557.001,A -85,B 0,C 180,E1 -25032.755,E2 -25032.755} C_VEL
LIN {X 0,Y 132.991,Z 552.58,A -85,B 0,C 180,E1 -25034.734,E2 -25034.734} C_VEL
LIN {X 0,Y 135.569,Z 544.492,A -85,B 0,C 180,E1 -25037.043,E2 -25037.043} C_VEL
LIN {X 0,Y 140.22,Z 528.79,A -85,B 0,C 180,E1 -25040.252,E2 -25040.252} C_VEL
LIN {X 0,Y 141.954,Z 526.027,A -85,B 0,C 180,E1 -25041.701,E2 -25041.701} C_VEL
LIN {X 0,Y 144.148,Z 520.753,A -85,B 0,C 180,E1 -25043.147,E2 -25043.147} C_VEL
LIN {X 0,Y 146.627,Z 512.734,A -85,B 0,C 180,E1 -25044.399,E2 -25044.399} C_VEL
LIN {X 0,Y 150.154,Z 499.675,A -85,B 0,C 180,E1 -25045.841,E2 -25045.841} C_VEL
LIN {X 0,Y 152.809,Z 496.348,A -85,B 0,C 180,E1 -25047.492,E2 -25047.492} C_VEL
LIN {X 0,Y 156.442,Z 492.711,A -85,B 0,C 180,E1 -25049.615,E2 -25049.615} C_VEL
LIN {X 0,Y 158.439,Z 490.55,A -85,B 0,C 180,E1 -25050.672,E2 -25050.672} C_VEL
LIN {X 0,Y 159.155,Z 491.253,A -85,B 0,C 180,E1 -25051.163,E2 -25051.163} C_VEL
LIN {X 0,Y 163.142,Z 498.626,A -85,B 0,C 180,E1 -25053.977,E2 -25053.977} C_VEL
LIN {X 0,Y 167.386,Z 507.656,A -85,B 0,C 180,E1 -25056.713,E2 -25056.713} C_VEL
LIN {X 0,Y 170.328,Z 514.729,A -85,B 0,C 180,E1 -25058.491,E2 -25058.491} C_VEL
LIN {X 0,Y 171.396,Z 532.49,A -85,B 0,C 180,E1 -25060.084,E2 -25060.084} C_VEL
LIN {X 0,Y 171.791,Z 541.559,A -85,B 0,C 180,E1 -25060.812,E2 -25060.812} C_VEL
LIN {X 0,Y 167.416,Z 601.894,A -85,B 0,C 180,E1 -25063.01,E2 -25063.01} C_VEL
LIN {X 0,Y 165.446,Z 614.81,A -85,B 0,C 180,E1 -25063.768,E2 -25063.768} C_VEL
LIN {X 0,Y 162.692,Z 627.488,A -85,B 0,C 180,E1 -25064.979,E2 -25064.979} C_VEL
LIN {X 0,Y 159.496,Z 638.823,A -85,B 0,C 180,E1 -25066.489,E2 -25066.489} C_VEL
LIN {X 0,Y 155.857,Z 649.22,A -85,B 0,C 180,E1 -25068.309,E2 -25068.309} C_VEL
LIN {X 0,Y 151.425,Z 659.863,A -85,B 0,C 180,E1 -25070.775,E2 -25070.775} C_VEL
LIN {X 0,Y 147.295,Z 668.555,A -85,B 0,C 180,E1 -25073.386,E2 -25073.386} C_VEL
LIN {X 0,Y 142.42,Z 678.003,A -85,B 0,C 180,E1 -25077.124,E2 -25077.124} C_VEL
LIN {X 0,Y 138.07,Z 685.5,A -85,B 0,C 180,E1 -25081.082,E2 -25081.082} C_VEL
LIN {X 0,Y 134.297,Z 691.514,A -85,B 0,C 180,E1 -25085.251,E2 -25085.251} C_VEL
LIN {X 0,Y 131.259,Z 696.268,A -85,B 0,C 180,E1 -25089.634,E2 -25089.634} C_VEL
LIN {X 0,Y 129.024,Z 699.903,A -85,B 0,C 180,E1 -25094.196,E2 -25094.196} C_VEL
LIN {X 0,Y 127.906,Z 701.774,A -85,B 0,C 180,E1 -25097.304,E2 -25097.304} C_VEL
LIN {X 0,Y 127.109,Z 703.197,A -85,B 0,C 180,E1 -25100.452,E2 -25100.452} C_VEL
LIN {X 0,Y 126.382,Z 704.81,A -85,B 0,C 180,E1 -25106.813,E2 -25106.813} C_VEL
LIN {X 0,Y 126.362,Z 705.04,A -85,B 0,C 180,E1 -25110,E2 -25110} C_VEL
LIN {X 0,Y 126.382,Z 704.839,A -85,B 0,C 180,E1 -25113.188,E2 -25113.188} C_VEL
LIN {X 0,Y 127.052,Z 703.265,A -85,B 0,C 180,E1 -25119.553,E2 -25119.553} C_VEL
LIN {X 0,Y 127.845,Z 701.88,A -85,B 0,C 180,E1 -25122.703,E2 -25122.703} C_VEL
LIN {X 0,Y 129.63,Z 698.974,A -85,B 0,C 180,E1 -25127.349,E2 -25127.349} C_VEL
LIN {X 0,Y 132.061,Z 695.026,A -85,B 0,C 180,E1 -25131.872,E2 -25131.872} C_VEL
LIN {X 0,Y 135.428,Z 689.908,A -85,B 0,C 180,E1 -25136.175,E2 -25136.175} C_VEL
LIN {X 0,Y 139.377,Z 683.459,A -85,B 0,C 180,E1 -25140.282,E2 -25140.282} C_VEL
LIN {X 0,Y 143.723,Z 675.735,A -85,B 0,C 180,E1 -25144.05,E2 -25144.05} C_VEL
LIN {X 0,Y 148.06,Z 667.243,A -85,B 0,C 180,E1 -25147.244,E2 -25147.244} C_VEL
LIN {X 0,Y 152.812,Z 657.12,A -85,B 0,C 180,E1 -25150.082,E2 -25150.082} C_VEL
LIN {X 0,Y 157.331,Z 645.734,A -85,B 0,C 180,E1 -25152.504,E2 -25152.504} C_VEL
LIN {X 0,Y 160.958,Z 634.461,A -85,B 0,C 180,E1 -25154.317,E2 -25154.317} C_VEL
LIN {X 0,Y 164.233,Z 621.638,A -85,B 0,C 180,E1 -25155.79,E2 -25155.79} C_VEL
LIN {X 0,Y 166.722,Z 608.447,A -85,B 0,C 180,E1 -25156.804,E2 -25156.804} C_VEL
LIN {X 0,Y 168.283,Z 593.795,A -85,B 0,C 180,E1 -25157.476,E2 -25157.476} C_VEL
LIN {X 0,Y 172.022,Z 540.041,A -85,B 0,C 180,E1 -25159.41,E2 -25159.41} C_VEL
LIN {X 0,Y 170.581,Z 515.534,A -85,B 0,C 180,E1 -25161.576,E2 -25161.576} C_VEL
LIN {X 0,Y 169.538,Z 512.447,A -85,B 0,C 180,E1 -25162.23,E2 -25162.23} C_VEL
LIN {X 0,Y 165.177,Z 502.636,A -85,B 0,C 180,E1 -25164.942,E2 -25164.942} C_VEL
LIN {X 0,Y 160.418,Z 493.34,A -85,B 0,C 180,E1 -25168.199,E2 -25168.199} C_VEL
LIN {X 0,Y 157.476,Z 487.861,A -85,B 0,C 180,E1 -25170.599,E2 -25170.599} C_VEL
LIN {X 0,Y 156.098,Z 482.709,A -85,B 0,C 180,E1 -25174.22,E2 -25174.22} C_VEL
LIN {X 0,Y 154.381,Z 477.416,A -85,B 0,C 180,E1 -25178.642,E2 -25178.642} C_VEL
LIN {X 0,Y 153.098,Z 473.614,A -85,B 0,C 180,E1 -25182.639,E2 -25182.639} C_VEL
LIN {X 0,Y 152.013,Z 470.613,A -85,B 0,C 180,E1 -25186.634,E2 -25186.634} C_VEL
LIN {X 0,Y 151.032,Z 467.453,A -85,B 0,C 180,E1 -25191.975,E2 -25191.975} C_VEL
LIN {X 0,Y 150.7,Z 464.856,A -85,B 0,C 180,E1 -25200,E2 -25200} C_VEL
LIN {X 0,Y 150.728,Z 464.868,A -85,B 0,C 180,E1 -25202.672,E2 -25202.672} C_VEL
LIN {X 0,Y 151.093,Z 466.056,A -85,B 0,C 180,E1 -25208.021,E2 -25208.021} C_VEL
LIN {X 0,Y 152.84,Z 469.033,A -85,B 0,C 180,E1 -25215.061,E2 -25215.061} C_VEL
LIN {X 0,Y 154.777,Z 472.391,A -85,B 0,C 180,E1 -25219.911,E2 -25219.911} C_VEL
LIN {X 0,Y 157.438,Z 477.473,A -85,B 0,C 180,E1 -25225.092,E2 -25225.092} C_VEL
LIN {X 0,Y 159.802,Z 482.422,A -85,B 0,C 180,E1 -25228.932,E2 -25228.932} C_VEL
LIN {X 0,Y 162.578,Z 488.334,A -85,B 0,C 180,E1 -25232.753,E2 -25232.753} C_VEL
LIN {X 0,Y 167.948,Z 496.911,A -85,B 0,C 180,E1 -25236.149,E2 -25236.149} C_VEL
LIN {X 0,Y 170.107,Z 500.586,A -85,B 0,C 180,E1 -25237.387,E2 -25237.387} C_VEL
LIN {X 0,Y 171.12,Z 526.516,A -85,B 0,C 180,E1 -25239.537,E2 -25239.537} C_VEL
LIN {X 0,Y 171.399,Z 544.69,A -85,B 0,C 180,E1 -25240.806,E2 -25240.806} C_VEL
LIN {X 0,Y 167.036,Z 604.563,A -85,B 0,C 180,E1 -25242.977,E2 -25242.977} C_VEL
LIN {X 0,Y 164.972,Z 617.919,A -85,B 0,C 180,E1 -25243.816,E2 -25243.816} C_VEL
LIN {X 0,Y 162.115,Z 630.374,A -85,B 0,C 180,E1 -25244.993,E2 -25244.993} C_VEL
LIN {X 0,Y 158.622,Z 642.324,A -85,B 0,C 180,E1 -25246.626,E2 -25246.626} C_VEL
LIN {X 0,Y 154.508,Z 653.667,A -85,B 0,C 180,E1 -25248.733,E2 -25248.733} C_VEL
LIN {X 0,Y 150.077,Z 663.894,A -85,B 0,C 180,E1 -25251.219,E2 -25251.219} C_VEL
LIN {X 0,Y 145.99,Z 672.257,A -85,B 0,C 180,E1 -25253.862,E2 -25253.862} C_VEL
LIN {X 0,Y 141.278,Z 681.013,A -85,B 0,C 180,E1 -25257.494,E2 -25257.494} C_VEL
LIN {X 0,Y 136.943,Z 688.561,A -85,B 0,C 180,E1 -25261.659,E2 -25261.659} C_VEL
LIN {X 0,Y 134.516,Z 692.558,A -85,B 0,C 180,E1 -25264.465,E2 -25264.465} C_VEL
LIN {X 0,Y 132.225,Z 695.223,A -85,B 0,C 180,E1 -25266.521,E2 -25266.521} C_VEL
LIN {X 0,Y 125.027,Z 700.294,A -85,B 0,C 180,E1 -25271.321,E2 -25271.321} C_VEL
LIN {X 0,Y 121.714,Z 702.569,A -85,B 0,C 180,E1 -25274.484,E2 -25274.484} C_VEL
LIN {X 0,Y 120.832,Z 703.516,A -85,B 0,C 180,E1 -25276.227,E2 -25276.227} C_VEL
LIN {X 0,Y 119.951,Z 705.098,A -85,B 0,C 180,E1 -25279.876,E2 -25279.876} C_VEL
LIN {X 0,Y 119.49,Z 706.093,A -85,B 0,C 180,E1 -25283.244,E2 -25283.244} C_VEL
LIN {X 0,Y 119.292,Z 706.7,A -85,B 0,C 180,E1 -25286.622,E2 -25286.622} C_VEL
LIN {X 0,Y 119.332,Z 706.912,A -85,B 0,C 180,E1 -25290,E2 -25290} C_VEL
LIN {X 0,Y 119.292,Z 706.684,A -85,B 0,C 180,E1 -25293.377,E2 -25293.377} C_VEL
LIN {X 0,Y 119.49,Z 706.066,A -85,B 0,C 180,E1 -25296.755,E2 -25296.755} C_VEL
LIN {X 0,Y 119.951,Z 705.06,A -85,B 0,C 180,E1 -25300.123,E2 -25300.123} C_VEL
LIN {X 0,Y 120.745,Z 703.631,A -85,B 0,C 180,E1 -25303.463,E2 -25303.463} C_VEL
LIN {X 0,Y 122.556,Z 700.667,A -85,B 0,C 180,E1 -25308.385,E2 -25308.385} C_VEL
LIN {X 0,Y 125.231,Z 696.646,A -85,B 0,C 180,E1 -25313.131,E2 -25313.131} C_VEL
LIN {X 0,Y 129.333,Z 690.451,A -85,B 0,C 180,E1 -25318.39,E2 -25318.39} C_VEL
LIN {X 0,Y 132.908,Z 684.911,A -85,B 0,C 180,E1 -25321.923,E2 -25321.923} C_VEL
LIN {X 0,Y 137.634,Z 676.776,A -85,B 0,C 180,E1 -25325.96,E2 -25325.96} C_VEL
LIN {X 0,Y 142.191,Z 668.425,A -85,B 0,C 180,E1 -25329.064,E2 -25329.064} C_VEL
LIN {X 0,Y 147.123,Z 658.101,A -85,B 0,C 180,E1 -25331.972,E2 -25331.972} C_VEL
LIN {X 0,Y 151.898,Z 646.483,A -85,B 0,C 180,E1 -25334.411,E2 -25334.411} C_VEL
LIN {X 0,Y 154.668,Z 639.887,A -85,B 0,C 180,E1 -25335.465,E2 -25335.465} C_VEL
LIN {X 0,Y 156.2,Z 639.372,A -85,B 0,C 180,E1 -25336.046,E2 -25336.046} C_VEL
LIN {X 0,Y 166.638,Z 637.53,A -85,B 0,C 180,E1 -25339.39,E2 -25339.39} C_VEL
LIN {X 0,Y 167.588,Z 636.935,A -85,B 0,C 180,E1 -25340.347,E2 -25340.347} C_VEL
LIN {X 0,Y 161.347,Z 636.003,A -85,B 0,C 180,E1 -25342.424,E2 -25342.424} C_VEL
LIN {X 0,Y 151.904,Z 633.405,A -85,B 0,C 180,E1 -25346.276,E2 -25346.276} C_VEL
LIN {X 0,Y 143.453,Z 629.463,A -85,B 0,C 180,E1 -25350.665,E2 -25350.665} C_VEL
LIN {X 0,Y 136.303,Z 624.066,A -85,B 0,C 180,E1 -25355.638,E2 -25355.638} C_VEL
LIN {X 0,Y 130.57,Z 617.166,A -85,B 0,C 180,E1 -25361.158,E2 -25361.158} C_VEL
LIN {X 0,Y 126.604,Z 608.663,A -85,B 0,C 180,E1 -25367.171,E2 -25367.171} C_VEL
LIN {X 0,Y 123.993,Z 600.801,A -85,B 0,C 180,E1 -25372.673,E2 -25372.673} C_VEL
LIN {X 0,Y 123.323,Z 596.866,A -85,B 0,C 180,E1 -25376.938,E2 -25376.938} C_VEL
LIN {X 0,Y 123.717,Z 592.327,A -85,B 0,C 180,E1 -25380.204,E2 -25380.204} C_VEL
LIN {X 0,Y 124.844,Z 585.705,A -85,B 0,C 180,E1 -25384.035,E2 -25384.035} C_VEL
LIN {X 0,Y 126.722,Z 577.404,A -85,B 0,C 180,E1 -25387.769,E2 -25387.769} C_VEL
LIN {X 0,Y 130.06,Z 565.41,A -85,B 0,C 180,E1 -25392.374,E2 -25392.374} C_VEL
LIN {X 0,Y 131.917,Z 562.095,A -85,B 0,C 180,E1 -25394.955,E2 -25394.955} C_VEL
LIN {X 0,Y 134.03,Z 556.873,A -85,B 0,C 180,E1 -25397.115,E2 -25397.115} C_VEL
LIN {X 0,Y 136.99,Z 548.324,A -85,B 0,C 180,E1 -25399.48,E2 -25399.48} C_VEL
LIN {X 0,Y 141.508,Z 534.007,A -85,B 0,C 180,E1 -25402.313,E2 -25402.313} C_VEL
LIN {X 0,Y 143.911,Z 529.867,A -85,B 0,C 180,E1 -25404.043,E2 -25404.043} C_VEL
LIN {X 0,Y 146.467,Z 523.765,A -85,B 0,C 180,E1 -25405.519,E2 -25405.519} C_VEL
LIN {X 0,Y 149.439,Z 514.521,A -85,B 0,C 180,E1 -25406.86,E2 -25406.86} C_VEL
LIN {X 0,Y 152.287,Z 504.495,A -85,B 0,C 180,E1 -25407.928,E2 -25407.928} C_VEL
LIN {X 0,Y 154.426,Z 501.98,A -85,B 0,C 180,E1 -25409.153,E2 -25409.153} C_VEL
LIN {X 0,Y 157.554,Z 498.915,A -85,B 0,C 180,E1 -25410.863,E2 -25410.863} C_VEL
LIN {X 0,Y 162.633,Z 509.567,A -85,B 0,C 180,E1 -25414.554,E2 -25414.554} C_VEL
LIN {X 0,Y 166.06,Z 517.925,A -85,B 0,C 180,E1 -25416.829,E2 -25416.829} C_VEL
LIN {X 0,Y 167.053,Z 538.426,A -85,B 0,C 180,E1 -25418.685,E2 -25418.685} C_VEL
LIN {X 0,Y 167.101,Z 543.553,A -85,B 0,C 180,E1 -25419.049,E2 -25419.049} C_VEL
LIN {X 0,Y 162.63,Z 602.28,A -85,B 0,C 180,E1 -25421.205,E2 -25421.205} C_VEL
LIN {X 0,Y 160.62,Z 614.836,A -85,B 0,C 180,E1 -25421.94,E2 -25421.94} C_VEL
LIN {X 0,Y 157.753,Z 627.525,A -85,B 0,C 180,E1 -25423.154,E2 -25423.154} C_VEL
LIN {X 0,Y 154.43,Z 638.865,A -85,B 0,C 180,E1 -25424.677,E2 -25424.677} C_VEL
LIN {X 0,Y 150.628,Z 649.267,A -85,B 0,C 180,E1 -25426.512,E2 -25426.512} C_VEL
LIN {X 0,Y 146.003,Z 659.913,A -85,B 0,C 180,E1 -25429.016,E2 -25429.016} C_VEL
LIN {X 0,Y 141.648,Z 668.607,A -85,B 0,C 180,E1 -25431.67,E2 -25431.67} C_VEL
LIN {X 0,Y 136.492,Z 678.056,A -85,B 0,C 180,E1 -25435.501,E2 -25435.501} C_VEL
LIN {X 0,Y 131.864,Z 685.554,A -85,B 0,C 180,E1 -25439.581,E2 -25439.581} C_VEL
LIN {X 0,Y 127.866,Z 691.568,A -85,B 0,C 180,E1 -25443.915,E2 -25443.915} C_VEL
LIN {X 0,Y 124.592,Z 696.323,A -85,B 0,C 180,E1 -25448.491,E2 -25448.491} C_VEL
LIN {X 0,Y 122.207,Z 699.957,A -85,B 0,C 180,E1 -25453.289,E2 -25453.289} C_VEL
LIN {X 0,Y 120.99,Z 701.828,A -85,B 0,C 180,E1 -25456.565,E2 -25456.565} C_VEL
LIN {X 0,Y 120.109,Z 703.252,A -85,B 0,C 180,E1 -25459.89,E2 -25459.89} C_VEL
LIN {X 0,Y 119.293,Z 704.864,A -85,B 0,C 180,E1 -25466.623,E2 -25466.623} C_VEL
LIN {X 0,Y 119.281,Z 705.094,A -85,B 0,C 180,E1 -25470,E2 -25470} C_VEL
LIN {X 0,Y 119.292,Z 704.893,A -85,B 0,C 180,E1 -25473.378,E2 -25473.378} C_VEL
LIN {X 0,Y 119.537,Z 704.298,A -85,B 0,C 180,E1 -25476.753,E2 -25476.753} C_VEL
LIN {X 0,Y 120.042,Z 703.318,A -85,B 0,C 180,E1 -25480.116,E2 -25480.116} C_VEL
LIN {X 0,Y 120.906,Z 701.933,A -85,B 0,C 180,E1 -25483.446,E2 -25483.446} C_VEL
LIN {X 0,Y 122.846,Z 699.027,A -85,B 0,C 180,E1 -25488.341,E2 -25488.341} C_VEL
LIN {X 0,Y 125.486,Z 695.078,A -85,B 0,C 180,E1 -25493.082,E2 -25493.082} C_VEL
LIN {X 0,Y 129.088,Z 689.959,A -85,B 0,C 180,E1 -25497.567,E2 -25497.567} C_VEL
LIN {X 0,Y 133.3,Z 683.508,A -85,B 0,C 180,E1 -25501.819,E2 -25501.819} C_VEL
LIN {X 0,Y 138.058,Z 675.491,A -85,B 0,C 180,E1 -25505.834,E2 -25505.834} C_VEL
LIN {X 0,Y 142.463,Z 667.288,A -85,B 0,C 180,E1 -25508.976,E2 -25508.976} C_VEL
LIN {X 0,Y 147.434,Z 657.161,A -85,B 0,C 180,E1 -25511.865,E2 -25511.865} C_VEL
LIN {X 0,Y 152.176,Z 645.77,A -85,B 0,C 180,E1 -25514.309,E2 -25514.309} C_VEL
LIN {X 0,Y 155.965,Z 634.489,A -85,B 0,C 180,E1 -25516.137,E2 -25516.137} C_VEL
LIN {X 0,Y 159.08,Z 622.894,A -85,B 0,C 180,E1 -25517.497,E2 -25517.497} C_VEL
LIN {X 0,Y 161.804,Z 609.482,A -85,B 0,C 180,E1 -25518.56,E2 -25518.56} C_VEL
LIN {X 0,Y 163.398,Z 596.081,A -85,B 0,C 180,E1 -25519.216,E2 -25519.216} C_VEL
LIN {X 0,Y 167.419,Z 541.162,A -85,B 0,C 180,E1 -25521.204,E2 -25521.204} C_VEL
LIN {X 0,Y 166.255,Z 518.379,A -85,B 0,C 180,E1 -25523.288,E2 -25523.288} C_VEL
LIN {X 0,Y 163.164,Z 510.609,A -85,B 0,C 180,E1 -25525.349,E2 -25525.349} C_VEL
LIN {X 0,Y 158.971,Z 501.751,A -85,B 0,C 180,E1 -25528.331,E2 -25528.331} C_VEL
LIN {X 0,Y 154.765,Z 493.687,A -85,B 0,C 180,E1 -25531.707,E2 -25531.707} C_VEL
LIN {X 0,Y 151.564,Z 487.923,A -85,B 0,C 180,E1 -25534.798,E2 -25534.798} C_VEL
LIN {X 0,Y 149.989,Z 482.515,A -85,B 0,C 180,E1 -25539.577,E2 -25539.577} C_VEL
LIN {X 0,Y 148.815,Z 478.901,A -85,B 0,C 180,E1 -25543.539,E2 -25543.539} C_VEL
LIN {X 0,Y 147.709,Z 475.152,A -85,B 0,C 180,E1 -25549.028,E2 -25549.028} C_VEL
LIN {X 0,Y 147.341,Z 473.693,A -85,B 0,C 180,E1 -25551.773,E2 -25551.773} C_VEL
LIN {X 0,Y 147.048,Z 471.007,A -85,B 0,C 180,E1 -25560,E2 -25560} C_VEL
LIN {X 0,Y 147.146,Z 471.033,A -85,B 0,C 180,E1 -25562.737,E2 -25562.737} C_VEL
LIN {X 0,Y 147.621,Z 472.318,A -85,B 0,C 180,E1 -25568.211,E2 -25568.211} C_VEL
LIN {X 0,Y 148.879,Z 474.523,A -85,B 0,C 180,E1 -25573.652,E2 -25573.652} C_VEL
LIN {X 0,Y 150.798,Z 477.947,A -85,B 0,C 180,E1 -25579.04,E2 -25579.04} C_VEL
LIN {X 0,Y 153.286,Z 482.9,A -85,B 0,C 180,E1 -25584.371,E2 -25584.371} C_VEL
LIN {X 0,Y 156.091,Z 488.71,A -85,B 0,C 180,E1 -25588.889,E2 -25588.889} C_VEL
LIN {X 0,Y 160.915,Z 495.984,A -85,B 0,C 180,E1 -25592.477,E2 -25592.477} C_VEL
LIN {X 0,Y 165.813,Z 504.062,A -85,B 0,C 180,E1 -25595.647,E2 -25595.647} C_VEL
LIN {X 0,Y 166.043,Z 505.605,A -85,B 0,C 180,E1 -25595.87,E2 -25595.87} C_VEL
LIN {X 0,Y 166.789,Z 536.546,A -85,B 0,C 180,E1 -25598.379,E2 -25598.379} C_VEL
LIN {X 0,Y 166.841,Z 544.937,A -85,B 0,C 180,E1 -25598.968,E2 -25598.968} C_VEL
LIN {X 0,Y 162.395,Z 603.701,A -85,B 0,C 180,E1 -25601.113,E2 -25601.113} C_VEL
LIN {X 0,Y 160.452,Z 616.445,A -85,B 0,C 180,E1 -25601.873,E2 -25601.873} C_VEL
LIN {X 0,Y 157.468,Z 629.253,A -85,B 0,C 180,E1 -25603.042,E2 -25603.042} C_VEL
LIN {X 0,Y 154.059,Z 640.65,A -85,B 0,C 180,E1 -25604.536,E2 -25604.536} C_VEL
LIN {X 0,Y 149.783,Z 652.357,A -85,B 0,C 180,E1 -25606.667,E2 -25606.667} C_VEL
LIN {X 0,Y 145.102,Z 662.797,A -85,B 0,C 180,E1 -25609.165,E2 -25609.165} C_VEL
LIN {X 0,Y 140.311,Z 672.211,A -85,B 0,C 180,E1 -25612.15,E2 -25612.15} C_VEL
LIN {X 0,Y 135.975,Z 679.902,A -85,B 0,C 180,E1 -25615.35,E2 -25615.35} C_VEL
LIN {X 0,Y 131.48,Z 687.404,A -85,B 0,C 180,E1 -25619.482,E2 -25619.482} C_VEL
LIN {X 0,Y 127.508,Z 693.43,A -85,B 0,C 180,E1 -25623.835,E2 -25623.835} C_VEL
LIN {X 0,Y 124.207,Z 698.186,A -85,B 0,C 180,E1 -25628.42,E2 -25628.42} C_VEL
LIN {X 0,Y 121.875,Z 701.818,A -85,B 0,C 180,E1 -25633.241,E2 -25633.241} C_VEL
LIN {X 0,Y 120.832,Z 703.516,A -85,B 0,C 180,E1 -25636.227,E2 -25636.227} C_VEL
LIN {X 0,Y 119.527,Z 704.85,A -85,B 0,C 180,E1 -25638.897,E2 -25638.897} C_VEL
LIN {X 0,Y 117.54,Z 705.829,A -85,B 0,C 180,E1 -25641.561,E2 -25641.561} C_VEL
LIN {X 0,Y 113.439,Z 706.797,A -85,B 0,C 180,E1 -25647.129,E2 -25647.129} C_VEL
LIN {X 0,Y 112.19,Z 706.787,A -85,B 0,C 180,E1 -25651.128,E2 -25651.128} C_VEL
LIN {X 0,Y 112.445,Z 706.012,A -85,B 0,C 180,E1 -25657.181,E2 -25657.181} C_VEL
LIN {X 0,Y 112.948,Z 705.006,A -85,B 0,C 180,E1 -25660.758,E2 -25660.758} C_VEL
LIN {X 0,Y 113.82,Z 703.576,A -85,B 0,C 180,E1 -25664.299,E2 -25664.299} C_VEL
LIN {X 0,Y 115.806,Z 700.613,A -85,B 0,C 180,E1 -25669.498,E2 -25669.498} C_VEL
LIN {X 0,Y 118.703,Z 696.592,A -85,B 0,C 180,E1 -25674.484,E2 -25674.484} C_VEL
LIN {X 0,Y 123.113,Z 690.397,A -85,B 0,C 180,E1 -25679.967,E2 -25679.967} C_VEL
LIN {X 0,Y 127.774,Z 683.526,A -85,B 0,C 180,E1 -25684.406,E2 -25684.406} C_VEL
LIN {X 0,Y 132.844,Z 675.168,A -85,B 0,C 180,E1 -25688.435,E2 -25688.435} C_VEL
LIN {X 0,Y 137.766,Z 666.455,A -85,B 0,C 180,E1 -25691.543,E2 -25691.543} C_VEL
LIN {X 0,Y 142.468,Z 656.897,A -85,B 0,C 180,E1 -25694.17,E2 -25694.17} C_VEL
LIN {X 0,Y 146.918,Z 646.439,A -85,B 0,C 180,E1 -25696.346,E2 -25696.346} C_VEL
LIN {X 0,Y 150.331,Z 638.484,A -85,B 0,C 180,E1 -25697.542,E2 -25697.542} C_VEL
LIN {X 0,Y 151.443,Z 638.081,A -85,B 0,C 180,E1 -25697.946,E2 -25697.946} C_VEL
LIN {X 0,Y 156.654,Z 637.473,A -85,B 0,C 180,E1 -25699.7,E2 -25699.7} C_VEL
LIN {X 0,Y 155.797,Z 636.792,A -85,B 0,C 180,E1 -25700.836,E2 -25700.836} C_VEL
LIN {X 0,Y 146.041,Z 633.648,A -85,B 0,C 180,E1 -25704.726,E2 -25704.726} C_VEL
LIN {X 0,Y 137.307,Z 629.17,A -85,B 0,C 180,E1 -25709.213,E2 -25709.213} C_VEL
LIN {X 0,Y 130.718,Z 624.523,A -85,B 0,C 180,E1 -25713.669,E2 -25713.669} C_VEL
LIN {X 0,Y 129.048,Z 623.667,A -85,B 0,C 180,E1 -25715.035,E2 -25715.035} C_VEL
LIN {X 0,Y 126.981,Z 623.092,A -85,B 0,C 180,E1 -25717.206,E2 -25717.206} C_VEL
LIN {X 0,Y 124.947,Z 621.428,A -85,B 0,C 180,E1 -25720.276,E2 -25720.276} C_VEL
LIN {X 0,Y 123.532,Z 618.897,A -85,B 0,C 180,E1 -25723.473,E2 -25723.473} C_VEL
LIN {X 0,Y 122.335,Z 613.1,A -85,B 0,C 180,E1 -25728.925,E2 -25728.925} C_VEL
LIN {X 0,Y 122.108,Z 606.406,A -85,B 0,C 180,E1 -25734.634,E2 -25734.634} C_VEL
LIN {X 0,Y 122.248,Z 603.198,A -85,B 0,C 180,E1 -25738.353,E2 -25738.353} C_VEL
LIN {X 0,Y 122.976,Z 598.643,A -85,B 0,C 180,E1 -25741.74,E2 -25741.74} C_VEL
LIN {X 0,Y 124.415,Z 591.832,A -85,B 0,C 180,E1 -25745.775,E2 -25745.775} C_VEL
LIN {X 0,Y 126.572,Z 583.562,A -85,B 0,C 180,E1 -25749.589,E2 -25749.589} C_VEL
LIN {X 0,Y 130.313,Z 571.207,A -85,B 0,C 180,E1 -25754.205,E2 -25754.205} C_VEL
LIN {X 0,Y 132.333,Z 567.915,A -85,B 0,C 180,E1 -25756.723,E2 -25756.723} C_VEL
LIN {X 0,Y 134.767,Z 562.481,A -85,B 0,C 180,E1 -25759.022,E2 -25759.022} C_VEL
LIN {X 0,Y 137.955,Z 554.125,A -85,B 0,C 180,E1 -25761.406,E2 -25761.406} C_VEL
LIN {X 0,Y 141.57,Z 543.474,A -85,B 0,C 180,E1 -25763.577,E2 -25763.577} C_VEL
LIN {X 0,Y 143.265,Z 538.582,A -85,B 0,C 180,E1 -25764.51,E2 -25764.51} C_VEL
LIN {X 0,Y 145.871,Z 534.082,A -85,B 0,C 180,E1 -25766.177,E2 -25766.177} C_VEL
LIN {X 0,Y 148.649,Z 527.8,A -85,B 0,C 180,E1 -25767.64,E2 -25767.64} C_VEL
LIN {X 0,Y 151.859,Z 518.404,A -85,B 0,C 180,E1 -25768.981,E2 -25768.981} C_VEL
LIN {X 0,Y 154.714,Z 508.898,A -85,B 0,C 180,E1 -25769.979,E2 -25769.979} C_VEL
LIN {X 0,Y 156.185,Z 507.607,A -85,B 0,C 180,E1 -25770.787,E2 -25770.787} C_VEL
LIN {X 0,Y 160.104,Z 516.457,A -85,B 0,C 180,E1 -25773.769,E2 -25773.769} C_VEL
LIN {X 0,Y 161.94,Z 521.427,A -85,B 0,C 180,E1 -25775.104,E2 -25775.104} C_VEL
LIN {X 0,Y 162.763,Z 542.978,A -85,B 0,C 180,E1 -25777.088,E2 -25777.088} C_VEL
LIN {X 0,Y 158.011,Z 602.653,A -85,B 0,C 180,E1 -25779.289,E2 -25779.289} C_VEL
LIN {X 0,Y 155.826,Z 615.584,A -85,B 0,C 180,E1 -25780.065,E2 -25780.065} C_VEL
LIN {X 0,Y 152.991,Z 627.563,A -85,B 0,C 180,E1 -25781.217,E2 -25781.217} C_VEL
LIN {X 0,Y 149.533,Z 638.908,A -85,B 0,C 180,E1 -25782.746,E2 -25782.746} C_VEL
LIN {X 0,Y 145.552,Z 649.313,A -85,B 0,C 180,E1 -25784.585,E2 -25784.585} C_VEL
LIN {X 0,Y 140.726,Z 659.962,A -85,B 0,C 180,E1 -25787.122,E2 -25787.122} C_VEL
LIN {X 0,Y 136.132,Z 668.658,A -85,B 0,C 180,E1 -25789.81,E2 -25789.81} C_VEL
LIN {X 0,Y 130.678,Z 678.109,A -85,B 0,C 180,E1 -25793.73,E2 -25793.73} C_VEL
LIN {X 0,Y 126.555,Z 684.486,A -85,B 0,C 180,E1 -25797.218,E2 -25797.218} C_VEL
LIN {X 0,Y 122.887,Z 689.775,A -85,B 0,C 180,E1 -25800.914,E2 -25800.914} C_VEL
LIN {X 0,Y 119.045,Z 694.942,A -85,B 0,C 180,E1 -25805.591,E2 -25805.591} C_VEL
LIN {X 0,Y 116.186,Z 698.938,A -85,B 0,C 180,E1 -25810.568,E2 -25810.568} C_VEL
LIN {X 0,Y 114.075,Z 701.883,A -85,B 0,C 180,E1 -25815.734,E2 -25815.734} C_VEL
LIN {X 0,Y 113.115,Z 703.306,A -85,B 0,C 180,E1 -25819.258,E2 -25819.258} C_VEL
LIN {X 0,Y 112.213,Z 704.918,A -85,B 0,C 180,E1 -25826.41,E2 -25826.41} C_VEL
LIN {X 0,Y 112.2,Z 705.148,A -85,B 0,C 180,E1 -25830,E2 -25830} C_VEL
LIN {X 0,Y 112.212,Z 704.946,A -85,B 0,C 180,E1 -25833.591,E2 -25833.591} C_VEL
LIN {X 0,Y 112.484,Z 704.351,A -85,B 0,C 180,E1 -25837.179,E2 -25837.179} C_VEL
LIN {X 0,Y 113.057,Z 703.372,A -85,B 0,C 180,E1 -25840.749,E2 -25840.749} C_VEL
LIN {X 0,Y 114.001,Z 701.986,A -85,B 0,C 180,E1 -25844.277,E2 -25844.277} C_VEL
LIN {X 0,Y 116.107,Z 699.079,A -85,B 0,C 180,E1 -25849.447,E2 -25849.447} C_VEL
LIN {X 0,Y 118.978,Z 695.13,A -85,B 0,C 180,E1 -25854.425,E2 -25854.425} C_VEL
LIN {X 0,Y 122.833,Z 690.009,A -85,B 0,C 180,E1 -25859.101,E2 -25859.101} C_VEL
LIN {X 0,Y 127.329,Z 683.557,A -85,B 0,C 180,E1 -25863.502,E2 -25863.502} C_VEL
LIN {X 0,Y 132.356,Z 675.539,A -85,B 0,C 180,E1 -25867.637,E2 -25867.637} C_VEL
LIN {X 0,Y 137.001,Z 667.333,A -85,B 0,C 180,E1 -25870.849,E2 -25870.849} C_VEL
LIN {X 0,Y 142.225,Z 657.202,A -85,B 0,C 180,E1 -25873.774,E2 -25873.774} C_VEL
LIN {X 0,Y 147.181,Z 645.806,A -85,B 0,C 180,E1 -25876.24,E2 -25876.24} C_VEL
LIN {X 0,Y 151.13,Z 634.517,A -85,B 0,C 180,E1 -25878.079,E2 -25878.079} C_VEL
LIN {X 0,Y 154.691,Z 621.668,A -85,B 0,C 180,E1 -25879.553,E2 -25879.553} C_VEL
LIN {X 0,Y 157.281,Z 608.825,A -85,B 0,C 180,E1 -25880.553,E2 -25880.553} C_VEL
LIN {X 0,Y 158.925,Z 595.215,A -85,B 0,C 180,E1 -25881.183,E2 -25881.183} C_VEL
LIN {X 0,Y 162.999,Z 542.009,A -85,B 0,C 180,E1 -25883.111,E2 -25883.111} C_VEL
LIN {X 0,Y 162.087,Z 521.263,A -85,B 0,C 180,E1 -25885.086,E2 -25885.086} C_VEL
LIN {X 0,Y 158.613,Z 512.68,A -85,B 0,C 180,E1 -25887.624,E2 -25887.624} C_VEL
LIN {X 0,Y 154.42,Z 503.731,A -85,B 0,C 180,E1 -25890.988,E2 -25890.988} C_VEL
LIN {X 0,Y 150.787,Z 496.882,A -85,B 0,C 180,E1 -25894.3,E2 -25894.3} C_VEL
LIN {X 0,Y 148.587,Z 493.017,A -85,B 0,C 180,E1 -25896.571,E2 -25896.571} C_VEL
LIN {X 0,Y 145.71,Z 487.874,A -85,B 0,C 180,E1 -25900.267,E2 -25900.267} C_VEL
LIN {X 0,Y 144.655,Z 484.248,A -85,B 0,C 180,E1 -25904.501,E2 -25904.501} C_VEL
LIN {X 0,Y 143.844,Z 481.384,A -85,B 0,C 180,E1 -25908.73,E2 -25908.73} C_VEL
LIN {X 0,Y 143.502,Z 479.872,A -85,B 0,C 180,E1 -25911.551,E2 -25911.551} C_VEL
LIN {X 0,Y 143.224,Z 477.954,A -85,B 0,C 180,E1 -25917.187,E2 -25917.187} C_VEL
LIN {X 0,Y 143.405,Z 477.152,A -85,B 0,C 180,E1 -25920,E2 -25920} C_VEL
LIN {X 0,Y 143.519,Z 477.159,A -85,B 0,C 180,E1 -25922.807,E2 -25922.807} C_VEL
LIN {X 0,Y 143.988,Z 478.512,A -85,B 0,C 180,E1 -25928.42,E2 -25928.42} C_VEL
LIN {X 0,Y 145.248,Z 480.824,A -85,B 0,C 180,E1 -25934,E2 -25934} C_VEL
LIN {X 0,Y 147.258,Z 484.518,A -85,B 0,C 180,E1 -25939.517,E2 -25939.517} C_VEL
LIN {X 0,Y 149.552,Z 488.86,A -85,B 0,C 180,E1 -25943.958,E2 -25943.958} C_VEL
LIN {X 0,Y 154.821,Z 496.465,A -85,B 0,C 180,E1 -25948.771,E2 -25948.771} C_VEL
LIN {X 0,Y 158.664,Z 502.614,A -85,B 0,C 180,E1 -25951.736,E2 -25951.736} C_VEL
LIN {X 0,Y 161.967,Z 508.326,A -85,B 0,C 180,E1 -25954.03,E2 -25954.03} C_VEL
LIN {X 0,Y 162.472,Z 540.534,A -85,B 0,C 180,E1 -25956.698,E2 -25956.698} C_VEL
LIN {X 0,Y 162.345,Z 546.641,A -85,B 0,C 180,E1 -25957.079,E2 -25957.079} C_VEL
LIN {X 0,Y 157.794,Z 604.045,A -85,B 0,C 180,E1 -25959.187,E2 -25959.187} C_VEL
LIN {X 0,Y 155.646,Z 617.171,A -85,B 0,C 180,E1 -25959.985,E2 -25959.985} C_VEL
LIN {X 0,Y 152.423,Z 630.329,A -85,B 0,C 180,E1 -25961.222,E2 -25961.222} C_VEL
LIN {X 0,Y 148.62,Z 642.257,A -85,B 0,C 180,E1 -25962.863,E2 -25962.863} C_VEL
LIN {X 0,Y 144.138,Z 653.588,A -85,B 0,C 180,E1 -25965.007,E2 -25965.007} C_VEL
LIN {X 0,Y 139.278,Z 663.808,A -85,B 0,C 180,E1 -25967.552,E2 -25967.552} C_VEL
LIN {X 0,Y 134.755,Z 672.165,A -85,B 0,C 180,E1 -25970.29,E2 -25970.29} C_VEL
LIN {X 0,Y 129.329,Z 681.198,A -85,B 0,C 180,E1 -25974.255,E2 -25974.255} C_VEL
LIN {X 0,Y 124.629,Z 688.461,A -85,B 0,C 180,E1 -25978.558,E2 -25978.558} C_VEL
LIN {X 0,Y 121.154,Z 693.379,A -85,B 0,C 180,E1 -25982.349,E2 -25982.349} C_VEL
LIN {X 0,Y 117.609,Z 698.134,A -85,B 0,C 180,E1 -25987.143,E2 -25987.143} C_VEL
LIN {X 0,Y 115.076,Z 701.765,A -85,B 0,C 180,E1 -25992.219,E2 -25992.219} C_VEL
LIN {X 0,Y 113.818,Z 703.636,A -85,B 0,C 180,E1 -25995.7,E2 -25995.7} C_VEL
LIN {X 0,Y 112.948,Z 705.044,A -85,B 0,C 180,E1 -25999.241,E2 -25999.241} C_VEL
LIN {X 0,Y 112.445,Z 706.039,A -85,B 0,C 180,E1 -26002.819,E2 -26002.819} C_VEL
LIN {X 0,Y 112.21,Z 706.647,A -85,B 0,C 180,E1 -26006.409,E2 -26006.409} C_VEL
LIN {X 0,Y 112.19,Z 706.787,A -85,B 0,C 180,E1 -26011.128,E2 -26011.128} C_VEL
LIN {X 0,Y 111.518,Z 706.572,A -85,B 0,C 180,E1 -26014.13,E2 -26014.13} C_VEL
LIN {X 0,Y 109.087,Z 705.588,A -85,B 0,C 180,E1 -26019.103,E2 -26019.103} C_VEL
LIN {X 0,Y 107.474,Z 704.297,A -85,B 0,C 180,E1 -26023.191,E2 -26023.191} C_VEL
LIN {X 0,Y 107.355,Z 703.017,A -85,B 0,C 180,E1 -26026.289,E2 -26026.289} C_VEL
LIN {X 0,Y 107.639,Z 702.476,A -85,B 0,C 180,E1 -26027.302,E2 -26027.302} C_VEL
LIN {X 0,Y 110.013,Z 699.326,A -85,B 0,C 180,E1 -26032.538,E2 -26032.538} C_VEL
LIN {X 0,Y 113.54,Z 694.938,A -85,B 0,C 180,E1 -26037.661,E2 -26037.661} C_VEL
LIN {X 0,Y 117.805,Z 689.343,A -85,B 0,C 180,E1 -26042.474,E2 -26042.474} C_VEL
LIN {X 0,Y 122.568,Z 682.567,A -85,B 0,C 180,E1 -26046.812,E2 -26046.812} C_VEL
LIN {X 0,Y 127.349,Z 675.116,A -85,B 0,C 180,E1 -26050.424,E2 -26050.424} C_VEL
LIN {X 0,Y 132.526,Z 666.404,A -85,B 0,C 180,E1 -26053.583,E2 -26053.583} C_VEL
LIN {X 0,Y 137.472,Z 656.85,A -85,B 0,C 180,E1 -26056.229,E2 -26056.229} C_VEL
LIN {X 0,Y 142.119,Z 646.394,A -85,B 0,C 180,E1 -26058.413,E2 -26058.413} C_VEL
LIN {X 0,Y 146.192,Z 636.988,A -85,B 0,C 180,E1 -26059.744,E2 -26059.744} C_VEL
LIN {X 0,Y 146.902,Z 636.543,A -85,B 0,C 180,E1 -26059.948,E2 -26059.948} C_VEL
LIN {X 0,Y 146.342,Z 636.096,A -85,B 0,C 180,E1 -26060.57,E2 -26060.57} C_VEL
LIN {X 0,Y 141.916,Z 635.029,A -85,B 0,C 180,E1 -26062.377,E2 -26062.377} C_VEL
LIN {X 0,Y 136.327,Z 634.97,A -85,B 0,C 180,E1 -26065.453,E2 -26065.453} C_VEL
LIN {X 0,Y 132.804,Z 634.07,A -85,B 0,C 180,E1 -26068.048,E2 -26068.048} C_VEL
LIN {X 0,Y 127.24,Z 630.702,A -85,B 0,C 180,E1 -26073.777,E2 -26073.777} C_VEL
LIN {X 0,Y 124.634,Z 629.748,A -85,B 0,C 180,E1 -26076.751,E2 -26076.751} C_VEL
LIN {X 0,Y 121.764,Z 627.32,A -85,B 0,C 180,E1 -26081.491,E2 -26081.491} C_VEL
LIN {X 0,Y 120.31,Z 623.203,A -85,B 0,C 180,E1 -26086.487,E2 -26086.487} C_VEL
LIN {X 0,Y 120.421,Z 612.677,A -85,B 0,C 180,E1 -26096.025,E2 -26096.025} C_VEL
LIN {X 0,Y 120.984,Z 609.264,A -85,B 0,C 180,E1 -26100,E2 -26100} C_VEL
LIN {X 0,Y 122.272,Z 604.272,A -85,B 0,C 180,E1 -26103.733,E2 -26103.733} C_VEL
LIN {X 0,Y 124.302,Z 597.187,A -85,B 0,C 180,E1 -26107.922,E2 -26107.922} C_VEL
LIN {X 0,Y 126.917,Z 588.525,A -85,B 0,C 180,E1 -26111.884,E2 -26111.884} C_VEL
LIN {X 0,Y 130.855,Z 576.871,A -85,B 0,C 180,E1 -26116.239,E2 -26116.239} C_VEL
LIN {X 0,Y 132.988,Z 573.507,A -85,B 0,C 180,E1 -26118.587,E2 -26118.587} C_VEL
LIN {X 0,Y 135.803,Z 567.729,A -85,B 0,C 180,E1 -26121.021,E2 -26121.021} C_VEL
LIN {X 0,Y 139.263,Z 559.384,A -85,B 0,C 180,E1 -26123.415,E2 -26123.415} C_VEL
LIN {X 0,Y 143.352,Z 548.158,A -85,B 0,C 180,E1 -26125.692,E2 -26125.692} C_VEL
LIN {X 0,Y 145.045,Z 543.361,A -85,B 0,C 180,E1 -26126.531,E2 -26126.531} C_VEL
LIN {X 0,Y 148.026,Z 538.297,A -85,B 0,C 180,E1 -26128.249,E2 -26128.249} C_VEL
LIN {X 0,Y 151.229,Z 531.316,A -85,B 0,C 180,E1 -26129.78,E2 -26129.78} C_VEL
LIN {X 0,Y 154.717,Z 521.535,A -85,B 0,C 180,E1 -26131.112,E2 -26131.112} C_VEL
LIN {X 0,Y 155.571,Z 518.836,A -85,B 0,C 180,E1 -26131.395,E2 -26131.395} C_VEL
LIN {X 0,Y 155.914,Z 519.049,A -85,B 0,C 180,E1 -26131.619,E2 -26131.619} C_VEL
LIN {X 0,Y 157.935,Z 524.357,A -85,B 0,C 180,E1 -26133.223,E2 -26133.223} C_VEL
LIN {X 0,Y 158.511,Z 544.03,A -85,B 0,C 180,E1 -26135.088,E2 -26135.088} C_VEL
LIN {X 0,Y 153.575,Z 603.043,A -85,B 0,C 180,E1 -26137.259,E2 -26137.259} C_VEL
LIN {X 0,Y 151.207,Z 616.332,A -85,B 0,C 180,E1 -26138.071,E2 -26138.071} C_VEL
LIN {X 0,Y 148.113,Z 628.684,A -85,B 0,C 180,E1 -26139.283,E2 -26139.283} C_VEL
LIN {X 0,Y 144.802,Z 638.951,A -85,B 0,C 180,E1 -26140.68,E2 -26140.68} C_VEL
LIN {X 0,Y 140.656,Z 649.359,A -85,B 0,C 180,E1 -26142.524,E2 -26142.524} C_VEL
LIN {X 0,Y 135.614,Z 660.011,A -85,B 0,C 180,E1 -26145.082,E2 -26145.082} C_VEL
LIN {X 0,Y 130.786,Z 668.709,A -85,B 0,C 180,E1 -26147.801,E2 -26147.801} C_VEL
LIN {X 0,Y 125.009,Z 678.161,A -85,B 0,C 180,E1 -26151.8,E2 -26151.8} C_VEL
LIN {X 0,Y 120.649,Z 684.539,A -85,B 0,C 180,E1 -26155.393,E2 -26155.393} C_VEL
LIN {X 0,Y 116.728,Z 689.829,A -85,B 0,C 180,E1 -26159.219,E2 -26159.219} C_VEL
LIN {X 0,Y 112.609,Z 694.996,A -85,B 0,C 180,E1 -26164.096,E2 -26164.096} C_VEL
LIN {X 0,Y 109.496,Z 698.993,A -85,B 0,C 180,E1 -26169.328,E2 -26169.328} C_VEL
LIN {X 0,Y 107.195,Z 701.937,A -85,B 0,C 180,E1 -26174.797,E2 -26174.797} C_VEL
LIN {X 0,Y 106.148,Z 703.36,A -85,B 0,C 180,E1 -26178.544,E2 -26178.544} C_VEL
LIN {X 0,Y 105.467,Z 704.359,A -85,B 0,C 180,E1 -26182.342,E2 -26182.342} C_VEL
LIN {X 0,Y 105.126,Z 704.972,A -85,B 0,C 180,E1 -26186.167,E2 -26186.167} C_VEL
LIN {X 0,Y 105.109,Z 705.202,A -85,B 0,C 180,E1 -26190.001,E2 -26190.001} C_VEL
LIN {X 0,Y 105.125,Z 705,A -85,B 0,C 180,E1 -26193.834,E2 -26193.834} C_VEL
LIN {X 0,Y 105.437,Z 704.405,A -85,B 0,C 180,E1 -26197.662,E2 -26197.662} C_VEL
LIN {X 0,Y 106.072,Z 703.425,A -85,B 0,C 180,E1 -26201.466,E2 -26201.466} C_VEL
LIN {X 0,Y 107.13,Z 702.039,A -85,B 0,C 180,E1 -26205.214,E2 -26205.214} C_VEL
LIN {X 0,Y 109.42,Z 699.132,A -85,B 0,C 180,E1 -26210.688,E2 -26210.688} C_VEL
LIN {X 0,Y 112.547,Z 695.182,A -85,B 0,C 180,E1 -26215.921,E2 -26215.921} C_VEL
LIN {X 0,Y 116.675,Z 690.06,A -85,B 0,C 180,E1 -26220.798,E2 -26220.798} C_VEL
LIN {X 0,Y 121.478,Z 683.606,A -85,B 0,C 180,E1 -26225.349,E2 -26225.349} C_VEL
LIN {X 0,Y 126.79,Z 675.586,A -85,B 0,C 180,E1 -26229.603,E2 -26229.603} C_VEL
LIN {X 0,Y 131.714,Z 667.378,A -85,B 0,C 180,E1 -26232.869,E2 -26232.869} C_VEL
LIN {X 0,Y 137.186,Z 657.243,A -85,B 0,C 180,E1 -26235.826,E2 -26235.826} C_VEL
LIN {X 0,Y 142.354,Z 645.843,A -85,B 0,C 180,E1 -26238.308,E2 -26238.308} C_VEL
LIN {X 0,Y 146.489,Z 634.544,A -85,B 0,C 180,E1 -26240.142,E2 -26240.142} C_VEL
LIN {X 0,Y 149.882,Z 622.926,A -85,B 0,C 180,E1 -26241.489,E2 -26241.489} C_VEL
LIN {X 0,Y 152.725,Z 609.793,A -85,B 0,C 180,E1 -26242.531,E2 -26242.531} C_VEL
LIN {X 0,Y 154.372,Z 597.396,A -85,B 0,C 180,E1 -26243.151,E2 -26243.151} C_VEL
LIN {X 0,Y 158.762,Z 542.936,A -85,B 0,C 180,E1 -26245.121,E2 -26245.121} C_VEL
LIN {X 0,Y 158.139,Z 524.642,A -85,B 0,C 180,E1 -26246.907,E2 -26246.907} C_VEL
LIN {X 0,Y 154.996,Z 516.707,A -85,B 0,C 180,E1 -26249.429,E2 -26249.429} C_VEL
LIN {X 0,Y 151.47,Z 508.772,A -85,B 0,C 180,E1 -26252.548,E2 -26252.548} C_VEL
LIN {X 0,Y 148.476,Z 502.752,A -85,B 0,C 180,E1 -26255.532,E2 -26255.532} C_VEL
LIN {X 0,Y 146.317,Z 498.841,A -85,B 0,C 180,E1 -26257.949,E2 -26257.949} C_VEL
LIN {X 0,Y 143.411,Z 493.681,A -85,B 0,C 180,E1 -26261.795,E2 -26261.795} C_VEL
LIN {X 0,Y 140.173,Z 488.115,A -85,B 0,C 180,E1 -26267.751,E2 -26267.751} C_VEL
LIN {X 0,Y 139.721,Z 486.108,A -85,B 0,C 180,E1 -26271.321,E2 -26271.321} C_VEL
LIN {X 0,Y 139.469,Z 484.023,A -85,B 0,C 180,E1 -26277.111,E2 -26277.111} C_VEL
LIN {X 0,Y 139.714,Z 483.248,A -85,B 0,C 180,E1 -26280,E2 -26280} C_VEL
LIN {X 0,Y 139.841,Z 483.241,A -85,B 0,C 180,E1 -26282.881,E2 -26282.881} C_VEL
LIN {X 0,Y 140.344,Z 484.686,A -85,B 0,C 180,E1 -26288.64,E2 -26288.64} C_VEL
LIN {X 0,Y 141.808,Z 487.243,A -85,B 0,C 180,E1 -26294.347,E2 -26294.347} C_VEL
LIN {X 0,Y 143.126,Z 489.29,A -85,B 0,C 180,E1 -26297.319,E2 -26297.319} C_VEL
LIN {X 0,Y 147.848,Z 495.577,A -85,B 0,C 180,E1 -26303.25,E2 -26303.25} C_VEL
LIN {X 0,Y 152.556,Z 502.686,A -85,B 0,C 180,E1 -26307.798,E2 -26307.798} C_VEL
LIN {X 0,Y 155.961,Z 508.378,A -85,B 0,C 180,E1 -26310.602,E2 -26310.602} C_VEL
LIN {X 0,Y 158.03,Z 512.046,A -85,B 0,C 180,E1 -26312.16,E2 -26312.16} C_VEL
LIN {X 0,Y 158.284,Z 537.099,A -85,B 0,C 180,E1 -26314.335,E2 -26314.335} C_VEL
LIN {X 0,Y 158.249,Z 545.934,A -85,B 0,C 180,E1 -26315.008,E2 -26315.008} C_VEL
LIN {X 0,Y 153.373,Z 604.392,A -85,B 0,C 180,E1 -26317.145,E2 -26317.145} C_VEL
LIN {X 0,Y 151.193,Z 617.164,A -85,B 0,C 180,E1 -26317.928,E2 -26317.928} C_VEL
LIN {X 0,Y 147.846,Z 630.306,A -85,B 0,C 180,E1 -26319.155,E2 -26319.155} C_VEL
LIN {X 0,Y 143.881,Z 642.223,A -85,B 0,C 180,E1 -26320.789,E2 -26320.789} C_VEL
LIN {X 0,Y 139.211,Z 653.549,A -85,B 0,C 180,E1 -26322.943,E2 -26322.943} C_VEL
LIN {X 0,Y 134.121,Z 663.765,A -85,B 0,C 180,E1 -26325.503,E2 -26325.503} C_VEL
LIN {X 0,Y 129.371,Z 672.119,A -85,B 0,C 180,E1 -26328.28,E2 -26328.28} C_VEL
LIN {X 0,Y 124.515,Z 679.806,A -85,B 0,C 180,E1 -26331.619,E2 -26331.619} C_VEL
LIN {X 0,Y 119.419,Z 687.341,A -85,B 0,C 180,E1 -26336.04,E2 -26336.04} C_VEL
LIN {X 0,Y 114.873,Z 693.327,A -85,B 0,C 180,E1 -26340.695,E2 -26340.695} C_VEL
LIN {X 0,Y 111.081,Z 698.082,A -85,B 0,C 180,E1 -26345.716,E2 -26345.716} C_VEL
LIN {X 0,Y 108.302,Z 701.712,A -85,B 0,C 180,E1 -26351.066,E2 -26351.066} C_VEL
LIN {X 0,Y 106.931,Z 703.583,A -85,B 0,C 180,E1 -26354.757,E2 -26354.757} C_VEL
LIN {X 0,Y 105.95,Z 704.99,A -85,B 0,C 180,E1 -26358.521,E2 -26358.521} C_VEL
LIN {X 0,Y 105.38,Z 705.986,A -85,B 0,C 180,E1 -26362.334,E2 -26362.334} C_VEL
LIN {X 0,Y 105.122,Z 706.593,A -85,B 0,C 180,E1 -26366.166,E2 -26366.166} C_VEL
LIN {X 0,Y 105.11,Z 706.742,A -85,B 0,C 180,E1 -26371.048,E2 -26371.048} C_VEL
LIN {X 0,Y 105.379,Z 705.958,A -85,B 0,C 180,E1 -26377.665,E2 -26377.665} C_VEL
LIN {X 0,Y 105.95,Z 704.951,A -85,B 0,C 180,E1 -26381.478,E2 -26381.478} C_VEL
LIN {X 0,Y 107.639,Z 702.476,A -85,B 0,C 180,E1 -26387.302,E2 -26387.302} C_VEL
LIN {X 0,Y 108.248,Z 700.907,A -85,B 0,C 180,E1 -26390.298,E2 -26390.298} C_VEL
LIN {X 0,Y 108.076,Z 697.763,A -85,B 0,C 180,E1 -26395.281,E2 -26395.281} C_VEL
LIN {X 0,Y 108.571,Z 694.026,A -85,B 0,C 180,E1 -26400.135,E2 -26400.135} C_VEL
LIN {X 0,Y 110.168,Z 691.332,A -85,B 0,C 180,E1 -26402.784,E2 -26402.784} C_VEL
LIN {X 0,Y 115.484,Z 684.505,A -85,B 0,C 180,E1 -26407.708,E2 -26407.708} C_VEL
LIN {X 0,Y 120.983,Z 676.619,A -85,B 0,C 180,E1 -26411.916,E2 -26411.916} C_VEL
LIN {X 0,Y 126.359,Z 668.273,A -85,B 0,C 180,E1 -26415.165,E2 -26415.165} C_VEL
LIN {X 0,Y 132.047,Z 657.955,A -85,B 0,C 180,E1 -26418.17,E2 -26418.17} C_VEL
LIN {X 0,Y 137.51,Z 646.349,A -85,B 0,C 180,E1 -26420.626,E2 -26420.626} C_VEL
LIN {X 0,Y 139.165,Z 642.495,A -85,B 0,C 180,E1 -26421.225,E2 -26421.225} C_VEL
LIN {X 0,Y 138.988,Z 641.385,A -85,B 0,C 180,E1 -26421.726,E2 -26421.726} C_VEL
LIN {X 0,Y 133.733,Z 641.313,A -85,B 0,C 180,E1 -26424.685,E2 -26424.685} C_VEL
LIN {X 0,Y 130.121,Z 640.528,A -85,B 0,C 180,E1 -26427.309,E2 -26427.309} C_VEL
LIN {X 0,Y 124.478,Z 637.405,A -85,B 0,C 180,E1 -26433.149,E2 -26433.149} C_VEL
LIN {X 0,Y 119.284,Z 634.397,A -85,B 0,C 180,E1 -26440.508,E2 -26440.508} C_VEL
LIN {X 0,Y 117.897,Z 631.87,A -85,B 0,C 180,E1 -26444.44,E2 -26444.44} C_VEL
LIN {X 0,Y 117.369,Z 627.247,A -85,B 0,C 180,E1 -26449.651,E2 -26449.651} C_VEL
LIN {X 0,Y 118.5,Z 618.858,A -85,B 0,C 180,E1 -26457.451,E2 -26457.451} C_VEL
LIN {X 0,Y 119.488,Z 615.325,A -85,B 0,C 180,E1 -26461.6,E2 -26461.6} C_VEL
LIN {X 0,Y 121.191,Z 610.528,A -85,B 0,C 180,E1 -26465.303,E2 -26465.303} C_VEL
LIN {X 0,Y 124.021,Z 603.08,A -85,B 0,C 180,E1 -26469.788,E2 -26469.788} C_VEL
LIN {X 0,Y 127.144,Z 594.39,A -85,B 0,C 180,E1 -26473.791,E2 -26473.791} C_VEL
LIN {X 0,Y 131.519,Z 582.526,A -85,B 0,C 180,E1 -26478.196,E2 -26478.196} C_VEL
LIN {X 0,Y 133.957,Z 578.796,A -85,B 0,C 180,E1 -26480.585,E2 -26480.585} C_VEL
LIN {X 0,Y 137.286,Z 572.375,A -85,B 0,C 180,E1 -26483.186,E2 -26483.186} C_VEL
LIN {X 0,Y 141.161,Z 563.574,A -85,B 0,C 180,E1 -26485.619,E2 -26485.619} C_VEL
LIN {X 0,Y 145.596,Z 552.11,A -85,B 0,C 180,E1 -26487.879,E2 -26487.879} C_VEL
LIN {X 0,Y 147.209,Z 547.795,A -85,B 0,C 180,E1 -26488.614,E2 -26488.614} C_VEL
LIN {X 0,Y 150.509,Z 542.225,A -85,B 0,C 180,E1 -26490.324,E2 -26490.324} C_VEL
LIN {X 0,Y 154.082,Z 534.646,A -85,B 0,C 180,E1 -26491.871,E2 -26491.871} C_VEL
LIN {X 0,Y 154.288,Z 534.145,A -85,B 0,C 180,E1 -26491.951,E2 -26491.951} C_VEL
LIN {X 0,Y 154.452,Z 544.995,A -85,B 0,C 180,E1 -26492.968,E2 -26492.968} C_VEL
LIN {X 0,Y 149.466,Z 602.317,A -85,B 0,C 180,E1 -26495.059,E2 -26495.059} C_VEL
LIN {X 0,Y 147.271,Z 614.913,A -85,B 0,C 180,E1 -26495.781,E2 -26495.781} C_VEL
LIN {X 0,Y 144.041,Z 627.635,A -85,B 0,C 180,E1 -26496.969,E2 -26496.969} C_VEL
LIN {X 0,Y 140.281,Z 638.993,A -85,B 0,C 180,E1 -26498.482,E2 -26498.482} C_VEL
LIN {X 0,Y 135.969,Z 649.406,A -85,B 0,C 180,E1 -26500.324,E2 -26500.324} C_VEL
LIN {X 0,Y 130.678,Z 660.061,A -85,B 0,C 180,E1 -26502.881,E2 -26502.881} C_VEL
LIN {X 0,Y 125.606,Z 668.76,A -85,B 0,C 180,E1 -26505.62,E2 -26505.62} C_VEL
LIN {X 0,Y 119.492,Z 678.214,A -85,B 0,C 180,E1 -26509.687,E2 -26509.687} C_VEL
LIN {X 0,Y 114.882,Z 684.593,A -85,B 0,C 180,E1 -26513.383,E2 -26513.383} C_VEL
LIN {X 0,Y 110.682,Z 689.883,A -85,B 0,C 180,E1 -26517.335,E2 -26517.335} C_VEL
LIN {X 0,Y 106.264,Z 695.05,A -85,B 0,C 180,E1 -26522.422,E2 -26522.422} C_VEL
LIN {X 0,Y 102.868,Z 699.047,A -85,B 0,C 180,E1 -26527.929,E2 -26527.929} C_VEL
LIN {X 0,Y 100.356,Z 701.992,A -85,B 0,C 180,E1 -26533.733,E2 -26533.733} C_VEL
LIN {X 0,Y 99.184,Z 703.415,A -85,B 0,C 180,E1 -26537.727,E2 -26537.727} C_VEL
LIN {X 0,Y 98.041,Z 705.027,A -85,B 0,C 180,E1 -26545.89,E2 -26545.89} C_VEL
LIN {X 0,Y 98.009,Z 705.256,A -85,B 0,C 180,E1 -26550.001,E2 -26550.001} C_VEL
LIN {X 0,Y 98.039,Z 705.054,A -85,B 0,C 180,E1 -26554.111,E2 -26554.111} C_VEL
LIN {X 0,Y 99.12,Z 703.479,A -85,B 0,C 180,E1 -26562.282,E2 -26562.282} C_VEL
LIN {X 0,Y 100.284,Z 702.092,A -85,B 0,C 180,E1 -26566.28,E2 -26566.28} C_VEL
LIN {X 0,Y 102.795,Z 699.185,A -85,B 0,C 180,E1 -26572.089,E2 -26572.089} C_VEL
LIN {X 0,Y 106.206,Z 695.233,A -85,B 0,C 180,E1 -26577.595,E2 -26577.595} C_VEL
LIN {X 0,Y 110.63,Z 690.11,A -85,B 0,C 180,E1 -26582.683,E2 -26582.683} C_VEL
LIN {X 0,Y 115.747,Z 683.655,A -85,B 0,C 180,E1 -26587.387,E2 -26587.387} C_VEL
LIN {X 0,Y 121.378,Z 675.633,A -85,B 0,C 180,E1 -26591.75,E2 -26591.75} C_VEL
LIN {X 0,Y 126.606,Z 667.423,A -85,B 0,C 180,E1 -26595.054,E2 -26595.054} C_VEL
LIN {X 0,Y 132.326,Z 657.285,A -85,B 0,C 180,E1 -26598.036,E2 -26598.036} C_VEL
LIN {X 0,Y 137.728,Z 645.879,A -85,B 0,C 180,E1 -26600.517,E2 -26600.517} C_VEL
LIN {X 0,Y 142.052,Z 634.572,A -85,B 0,C 180,E1 -26602.336,E2 -26602.336} C_VEL
LIN {X 0,Y 145.57,Z 622.944,A -85,B 0,C 180,E1 -26603.675,E2 -26603.675} C_VEL
LIN {X 0,Y 148.476,Z 609.957,A -85,B 0,C 180,E1 -26604.697,E2 -26604.697} C_VEL
LIN {X 0,Y 150.304,Z 596.658,A -85,B 0,C 180,E1 -26605.332,E2 -26605.332} C_VEL
LIN {X 0,Y 154.716,Z 543.781,A -85,B 0,C 180,E1 -26607.253,E2 -26607.253} C_VEL
LIN {X 0,Y 154.364,Z 528.109,A -85,B 0,C 180,E1 -26608.809,E2 -26608.809} C_VEL
LIN {X 0,Y 151.54,Z 520.59,A -85,B 0,C 180,E1 -26611.333,E2 -26611.333} C_VEL
LIN {X 0,Y 148.262,Z 512.95,A -85,B 0,C 180,E1 -26614.564,E2 -26614.564} C_VEL
LIN {X 0,Y 144.971,Z 506.064,A -85,B 0,C 180,E1 -26618.326,E2 -26618.326} C_VEL
LIN {X 0,Y 141.837,Z 500.223,A -85,B 0,C 180,E1 -26622.704,E2 -26622.704} C_VEL
LIN {X 0,Y 138.849,Z 494.85,A -85,B 0,C 180,E1 -26628.504,E2 -26628.504} C_VEL
LIN {X 0,Y 137.145,Z 491.76,A -85,B 0,C 180,E1 -26634.117,E2 -26634.117} C_VEL
LIN {X 0,Y 136.652,Z 489.714,A -85,B 0,C 180,E1 -26640,E2 -26640} C_VEL
LIN {X 0,Y 136.901,Z 489.872,A -85,B 0,C 180,E1 -26643.679,E2 -26643.679} C_VEL
LIN {X 0,Y 138.656,Z 492.298,A -85,B 0,C 180,E1 -26650.588,E2 -26650.588} C_VEL
LIN {X 0,Y 141.389,Z 495.54,A -85,B 0,C 180,E1 -26656.051,E2 -26656.051} C_VEL
LIN {X 0,Y 145.753,Z 501.636,A -85,B 0,C 180,E1 -26662.037,E2 -26662.037} C_VEL
LIN {X 0,Y 150.203,Z 508.699,A -85,B 0,C 180,E1 -26666.673,E2 -26666.673} C_VEL
LIN {X 0,Y 153.336,Z 514.19,A -85,B 0,C 180,E1 -26669.441,E2 -26669.441} C_VEL
LIN {X 0,Y 154.33,Z 515.934,A -85,B 0,C 180,E1 -26670.25,E2 -26670.25} C_VEL
LIN {X 0,Y 154.286,Z 544.583,A -85,B 0,C 180,E1 -26672.726,E2 -26672.726} C_VEL
LIN {X 0,Y 153.67,Z 553.263,A -85,B 0,C 180,E1 -26673.101,E2 -26673.101} C_VEL
LIN {X 0,Y 149.308,Z 603.595,A -85,B 0,C 180,E1 -26674.945,E2 -26674.945} C_VEL
LIN {X 0,Y 147.121,Z 616.424,A -85,B 0,C 180,E1 -26675.698,E2 -26675.698} C_VEL
LIN {X 0,Y 143.795,Z 629.186,A -85,B 0,C 180,E1 -26676.837,E2 -26676.837} C_VEL
LIN {X 0,Y 139.96,Z 640.555,A -85,B 0,C 180,E1 -26678.315,E2 -26678.315} C_VEL
LIN {X 0,Y 135.086,Z 652.241,A -85,B 0,C 180,E1 -26680.457,E2 -26680.457} C_VEL
LIN {X 0,Y 129.754,Z 662.669,A -85,B 0,C 180,E1 -26683.01,E2 -26683.01} C_VEL
LIN {X 0,Y 124.161,Z 672.073,A -85,B 0,C 180,E1 -26686.099,E2 -26686.099} C_VEL
LIN {X 0,Y 119.011,Z 679.757,A -85,B 0,C 180,E1 -26689.489,E2 -26689.489} C_VEL
LIN {X 0,Y 113.605,Z 687.255,A -85,B 0,C 180,E1 -26694.005,E2 -26694.005} C_VEL
LIN {X 0,Y 108.699,Z 693.276,A -85,B 0,C 180,E1 -26698.852,E2 -26698.852} C_VEL
LIN {X 0,Y 104.634,Z 698.03,A -85,B 0,C 180,E1 -26704.113,E2 -26704.113} C_VEL
LIN {X 0,Y 101.587,Z 701.659,A -85,B 0,C 180,E1 -26709.762,E2 -26709.762} C_VEL
LIN {X 0,Y 100.085,Z 703.53,A -85,B 0,C 180,E1 -26713.686,E2 -26713.686} C_VEL
LIN {X 0,Y 98.984,Z 704.937,A -85,B 0,C 180,E1 -26717.701,E2 -26717.701} C_VEL
LIN {X 0,Y 98.332,Z 705.932,A -85,B 0,C 180,E1 -26721.781,E2 -26721.781} C_VEL
LIN {X 0,Y 98.034,Z 706.539,A -85,B 0,C 180,E1 -26725.888,E2 -26725.888} C_VEL
LIN {X 0,Y 98.077,Z 706.75,A -85,B 0,C 180,E1 -26729.999,E2 -26729.999} C_VEL
LIN {X 0,Y 98.034,Z 706.521,A -85,B 0,C 180,E1 -26734.111,E2 -26734.111} C_VEL
LIN {X 0,Y 98.332,Z 705.903,A -85,B 0,C 180,E1 -26738.218,E2 -26738.218} C_VEL
LIN {X 0,Y 98.985,Z 704.897,A -85,B 0,C 180,E1 -26742.298,E2 -26742.298} C_VEL
LIN {X 0,Y 100.712,Z 702.61,A -85,B 0,C 180,E1 -26748.112,E2 -26748.112} C_VEL
LIN {X 0,Y 103.465,Z 699.272,A -85,B 0,C 180,E1 -26754.051,E2 -26754.051} C_VEL
LIN {X 0,Y 107.287,Z 694.884,A -85,B 0,C 180,E1 -26759.426,E2 -26759.426} C_VEL
LIN {X 0,Y 110.168,Z 691.332,A -85,B 0,C 180,E1 -26762.784,E2 -26762.784} C_VEL
LIN {X 0,Y 111.915,Z 688.494,A -85,B 0,C 180,E1 -26765.307,E2 -26765.307} C_VEL
LIN {X 0,Y 113.499,Z 683.421,A -85,B 0,C 180,E1 -26769.575,E2 -26769.575} C_VEL
LIN {X 0,Y 115.457,Z 677.714,A -85,B 0,C 180,E1 -26773.513,E2 -26773.513} C_VEL
LIN {X 0,Y 117.676,Z 673.866,A -85,B 0,C 180,E1 -26775.429,E2 -26775.429} C_VEL
LIN {X 0,Y 123.781,Z 664.377,A -85,B 0,C 180,E1 -26778.79,E2 -26778.79} C_VEL
LIN {X 0,Y 129.222,Z 654.504,A -85,B 0,C 180,E1 -26781.348,E2 -26781.348} C_VEL
LIN {X 0,Y 132.439,Z 647.708,A -85,B 0,C 180,E1 -26782.749,E2 -26782.749} C_VEL
LIN {X 0,Y 127.174,Z 646.738,A -85,B 0,C 180,E1 -26786.452,E2 -26786.452} C_VEL
LIN {X 0,Y 118.917,Z 642.669,A -85,B 0,C 180,E1 -26795.562,E2 -26795.562} C_VEL
LIN {X 0,Y 115.281,Z 639.757,A -85,B 0,C 180,E1 -26802.253,E2 -26802.253} C_VEL
LIN {X 0,Y 114.295,Z 636.116,A -85,B 0,C 180,E1 -26807.572,E2 -26807.572} C_VEL
LIN {X 0,Y 114.744,Z 631.103,A -85,B 0,C 180,E1 -26812.964,E2 -26812.964} C_VEL
LIN {X 0,Y 116.178,Z 625.481,A -85,B 0,C 180,E1 -26818.267,E2 -26818.267} C_VEL
LIN {X 0,Y 117.861,Z 621.102,A -85,B 0,C 180,E1 -26823.419,E2 -26823.419} C_VEL
LIN {X 0,Y 120.137,Z 616.191,A -85,B 0,C 180,E1 -26827.29,E2 -26827.29} C_VEL
LIN {X 0,Y 123.617,Z 608.887,A -85,B 0,C 180,E1 -26831.686,E2 -26831.686} C_VEL
LIN {X 0,Y 127.426,Z 600.258,A -85,B 0,C 180,E1 -26835.7,E2 -26835.7} C_VEL
LIN {X 0,Y 132.218,Z 588.289,A -85,B 0,C 180,E1 -26840.01,E2 -26840.01} C_VEL
LIN {X 0,Y 134.995,Z 584.234,A -85,B 0,C 180,E1 -26842.478,E2 -26842.478} C_VEL
LIN {X 0,Y 138.765,Z 577.411,A -85,B 0,C 180,E1 -26845.177,E2 -26845.177} C_VEL
LIN {X 0,Y 142.954,Z 568.491,A -85,B 0,C 180,E1 -26847.603,E2 -26847.603} C_VEL
LIN {X 0,Y 147.749,Z 556.782,A -85,B 0,C 180,E1 -26849.866,E2 -26849.866} C_VEL
LIN {X 0,Y 149.565,Z 552.192,A -85,B 0,C 180,E1 -26850.634,E2 -26850.634} C_VEL
LIN {X 0,Y 150.096,Z 551.422,A -85,B 0,C 180,E1 -26850.904,E2 -26850.904} C_VEL
LIN {X 0,Y 145.438,Z 602.915,A -85,B 0,C 180,E1 -26852.8,E2 -26852.8} C_VEL
LIN {X 0,Y 143.071,Z 615.663,A -85,B 0,C 180,E1 -26853.535,E2 -26853.535} C_VEL
LIN {X 0,Y 139.57,Z 628.757,A -85,B 0,C 180,E1 -26854.774,E2 -26854.774} C_VEL
LIN {X 0,Y 135.35,Z 640.695,A -85,B 0,C 180,E1 -26856.406,E2 -26856.406} C_VEL
LIN {X 0,Y 130.23,Z 652.003,A -85,B 0,C 180,E1 -26858.51,E2 -26858.51} C_VEL
LIN {X 0,Y 124.752,Z 662.203,A -85,B 0,C 180,E1 -26861.106,E2 -26861.106} C_VEL
LIN {X 0,Y 119.496,Z 670.561,A -85,B 0,C 180,E1 -26863.907,E2 -26863.907} C_VEL
LIN {X 0,Y 114.158,Z 678.266,A -85,B 0,C 180,E1 -26867.375,E2 -26867.375} C_VEL
LIN {X 0,Y 108.298,Z 685.767,A -85,B 0,C 180,E1 -26871.939,E2 -26871.939} C_VEL
LIN {X 0,Y 103.097,Z 691.784,A -85,B 0,C 180,E1 -26876.952,E2 -26876.952} C_VEL
LIN {X 0,Y 98.664,Z 696.54,A -85,B 0,C 180,E1 -26882.419,E2 -26882.419} C_VEL
LIN {X 0,Y 95.274,Z 700.175,A -85,B 0,C 180,E1 -26888.357,E2 -26888.357} C_VEL
LIN {X 0,Y 93.535,Z 702.046,A -85,B 0,C 180,E1 -26892.51,E2 -26892.51} C_VEL
LIN {X 0,Y 92.256,Z 703.469,A -85,B 0,C 180,E1 -26896.79,E2 -26896.79} C_VEL
LIN {X 0,Y 90.952,Z 705.081,A -85,B 0,C 180,E1 -26905.569,E2 -26905.569} C_VEL
LIN {X 0,Y 90.918,Z 705.31,A -85,B 0,C 180,E1 -26910.001,E2 -26910.001} C_VEL
LIN {X 0,Y 90.949,Z 705.108,A -85,B 0,C 180,E1 -26914.433,E2 -26914.433} C_VEL
LIN {X 0,Y 91.361,Z 704.513,A -85,B 0,C 180,E1 -26918.851,E2 -26918.851} C_VEL
LIN {X 0,Y 92.177,Z 703.532,A -85,B 0,C 180,E1 -26923.223,E2 -26923.223} C_VEL
LIN {X 0,Y 93.471,Z 702.145,A -85,B 0,C 180,E1 -26927.504,E2 -26927.504} C_VEL
LIN {X 0,Y 96.217,Z 699.237,A -85,B 0,C 180,E1 -26933.688,E2 -26933.688} C_VEL
LIN {X 0,Y 99.972,Z 695.285,A -85,B 0,C 180,E1 -26939.479,E2 -26939.479} C_VEL
LIN {X 0,Y 104.717,Z 690.161,A -85,B 0,C 180,E1 -26944.784,E2 -26944.784} C_VEL
LIN {X 0,Y 110.175,Z 683.704,A -85,B 0,C 180,E1 -26949.636,E2 -26949.636} C_VEL
LIN {X 0,Y 116.155,Z 675.681,A -85,B 0,C 180,E1 -26954.093,E2 -26954.093} C_VEL
LIN {X 0,Y 121.689,Z 667.468,A -85,B 0,C 180,E1 -26957.423,E2 -26957.423} C_VEL
LIN {X 0,Y 127.69,Z 657.326,A -85,B 0,C 180,E1 -26960.405,E2 -26960.405} C_VEL
LIN {X 0,Y 133.331,Z 645.916,A -85,B 0,C 180,E1 -26962.87,E2 -26962.87} C_VEL
LIN {X 0,Y 137.826,Z 634.6,A -85,B 0,C 180,E1 -26964.674,E2 -26964.674} C_VEL
LIN {X 0,Y 141.824,Z 621.718,A -85,B 0,C 180,E1 -26966.104,E2 -26966.104} C_VEL
LIN {X 0,Y 144.739,Z 608.58,A -85,B 0,C 180,E1 -26967.081,E2 -26967.081} C_VEL
LIN {X 0,Y 146.57,Z 594.5,A -85,B 0,C 180,E1 -26967.699,E2 -26967.699} C_VEL
LIN {X 0,Y 150.91,Z 545.256,A -85,B 0,C 180,E1 -26969.431,E2 -26969.431} C_VEL
LIN {X 0,Y 150.711,Z 531.206,A -85,B 0,C 180,E1 -26970.878,E2 -26970.878} C_VEL
LIN {X 0,Y 147.257,Z 521.998,A -85,B 0,C 180,E1 -26974.378,E2 -26974.378} C_VEL
LIN {X 0,Y 144.286,Z 515.038,A -85,B 0,C 180,E1 -26977.83,E2 -26977.83} C_VEL
LIN {X 0,Y 142.513,Z 511.279,A -85,B 0,C 180,E1 -26980.181,E2 -26980.181} C_VEL
LIN {X 0,Y 140.097,Z 506.404,A -85,B 0,C 180,E1 -26983.984,E2 -26983.984} C_VEL
LIN {X 0,Y 137.549,Z 501.432,A -85,B 0,C 180,E1 -26989.512,E2 -26989.512} C_VEL
LIN {X 0,Y 136.08,Z 498.436,A -85,B 0,C 180,E1 -26995.186,E2 -26995.186} C_VEL
LIN {X 0,Y 135.78,Z 496.821,A -85,B 0,C 180,E1 -27000,E2 -27000} C_VEL
LIN {X 0,Y 136.012,Z 496.915,A -85,B 0,C 180,E1 -27003.518,E2 -27003.518} C_VEL
LIN {X 0,Y 137.653,Z 499.301,A -85,B 0,C 180,E1 -27010.294,E2 -27010.294} C_VEL
LIN {X 0,Y 140.08,Z 502.36,A -85,B 0,C 180,E1 -27015.411,E2 -27015.411} C_VEL
LIN {X 0,Y 144.004,Z 508.152,A -85,B 0,C 180,E1 -27021.143,E2 -27021.143} C_VEL
LIN {X 0,Y 147.986,Z 514.821,A -85,B 0,C 180,E1 -27025.586,E2 -27025.586} C_VEL
LIN {X 0,Y 150.747,Z 519.954,A -85,B 0,C 180,E1 -27028.216,E2 -27028.216} C_VEL
LIN {X 0,Y 150.604,Z 539.794,A -85,B 0,C 180,E1 -27030.025,E2 -27030.025} C_VEL
LIN {X 0,Y 150.403,Z 547.742,A -85,B 0,C 180,E1 -27030.63,E2 -27030.63} C_VEL
LIN {X 0,Y 145.327,Z 603.978,A -85,B 0,C 180,E1 -27032.671,E2 -27032.671} C_VEL
LIN {X 0,Y 142.916,Z 617.148,A -85,B 0,C 180,E1 -27033.44,E2 -27033.44} C_VEL
LIN {X 0,Y 139.332,Z 630.26,A -85,B 0,C 180,E1 -27034.631,E2 -27034.631} C_VEL
LIN {X 0,Y 135.018,Z 642.155,A -85,B 0,C 180,E1 -27036.213,E2 -27036.213} C_VEL
LIN {X 0,Y 129.962,Z 653.47,A -85,B 0,C 180,E1 -27038.359,E2 -27038.359} C_VEL
LIN {X 0,Y 124.391,Z 663.679,A -85,B 0,C 180,E1 -27040.914,E2 -27040.914} C_VEL
LIN {X 0,Y 119.132,Z 672.027,A -85,B 0,C 180,E1 -27043.724,E2 -27043.724} C_VEL
LIN {X 0,Y 112.661,Z 681.05,A -85,B 0,C 180,E1 -27047.885,E2 -27047.885} C_VEL
LIN {X 0,Y 107.282,Z 687.977,A -85,B 0,C 180,E1 -27052.344,E2 -27052.344} C_VEL
LIN {X 0,Y 102.655,Z 693.225,A -85,B 0,C 180,E1 -27056.79,E2 -27056.79} C_VEL
LIN {X 0,Y 98.284,Z 697.978,A -85,B 0,C 180,E1 -27062.302,E2 -27062.302} C_VEL
LIN {X 0,Y 94.911,Z 701.606,A -85,B 0,C 180,E1 -27068.269,E2 -27068.269} C_VEL
LIN {X 0,Y 93.269,Z 703.477,A -85,B 0,C 180,E1 -27072.457,E2 -27072.457} C_VEL
LIN {X 0,Y 92.053,Z 704.883,A -85,B 0,C 180,E1 -27076.759,E2 -27076.759} C_VEL
LIN {X 0,Y 91.31,Z 705.878,A -85,B 0,C 180,E1 -27081.144,E2 -27081.144} C_VEL
LIN {X 0,Y 90.943,Z 706.485,A -85,B 0,C 180,E1 -27085.567,E2 -27085.567} C_VEL
LIN {X 0,Y 90.977,Z 706.696,A -85,B 0,C 180,E1 -27089.999,E2 -27089.999} C_VEL
LIN {X 0,Y 90.943,Z 706.467,A -85,B 0,C 180,E1 -27094.432,E2 -27094.432} C_VEL
LIN {X 0,Y 91.31,Z 705.849,A -85,B 0,C 180,E1 -27098.855,E2 -27098.855} C_VEL
LIN {X 0,Y 92.053,Z 704.843,A -85,B 0,C 180,E1 -27103.24,E2 -27103.24} C_VEL
LIN {X 0,Y 93.27,Z 703.412,A -85,B 0,C 180,E1 -27107.541,E2 -27107.541} C_VEL
LIN {X 0,Y 95.891,Z 700.449,A -85,B 0,C 180,E1 -27113.772,E2 -27113.772} C_VEL
LIN {X 0,Y 99.661,Z 696.429,A -85,B 0,C 180,E1 -27119.579,E2 -27119.579} C_VEL
LIN {X 0,Y 104.3,Z 691.234,A -85,B 0,C 180,E1 -27124.942,E2 -27124.942} C_VEL
LIN {X 0,Y 109.748,Z 684.699,A -85,B 0,C 180,E1 -27129.82,E2 -27129.82} C_VEL
LIN {X 0,Y 115.785,Z 676.567,A -85,B 0,C 180,E1 -27134.269,E2 -27134.269} C_VEL
LIN {X 0,Y 117.676,Z 673.866,A -85,B 0,C 180,E1 -27135.429,E2 -27135.429} C_VEL
LIN {X 0,Y 119.027,Z 671.222,A -85,B 0,C 180,E1 -27136.719,E2 -27136.719} C_VEL
LIN {X 0,Y 119.862,Z 667.017,A -85,B 0,C 180,E1 -27139.233,E2 -27139.233} C_VEL
LIN {X 0,Y 120.742,Z 662.583,A -85,B 0,C 180,E1 -27141.625,E2 -27141.625} C_VEL
LIN {X 0,Y 122.076,Z 659.565,A -85,B 0,C 180,E1 -27142.68,E2 -27142.68} C_VEL
LIN {X 0,Y 125.274,Z 653.721,A -85,B 0,C 180,E1 -27144.06,E2 -27144.06} C_VEL
LIN {X 0,Y 124.872,Z 652.886,A -85,B 0,C 180,E1 -27144.768,E2 -27144.768} C_VEL
LIN {X 0,Y 120.744,Z 651.599,A -85,B 0,C 180,E1 -27148.409,E2 -27148.409} C_VEL
LIN {X 0,Y 111.876,Z 646.156,A -85,B 0,C 180,E1 -27161.694,E2 -27161.694} C_VEL
LIN {X 0,Y 110.771,Z 642.971,A -85,B 0,C 180,E1 -27167.17,E2 -27167.17} C_VEL
LIN {X 0,Y 111.281,Z 638.465,A -85,B 0,C 180,E1 -27172.744,E2 -27172.744} C_VEL
LIN {X 0,Y 113.769,Z 631.275,A -85,B 0,C 180,E1 -27180,E2 -27180} C_VEL
LIN {X 0,Y 116.023,Z 626.88,A -85,B 0,C 180,E1 -27185.213,E2 -27185.213} C_VEL
LIN {X 0,Y 118.854,Z 621.949,A -85,B 0,C 180,E1 -27189.175,E2 -27189.175} C_VEL
LIN {X 0,Y 123.209,Z 614.393,A -85,B 0,C 180,E1 -27193.756,E2 -27193.756} C_VEL
LIN {X 0,Y 127.74,Z 605.848,A -85,B 0,C 180,E1 -27197.717,E2 -27197.717} C_VEL
LIN {X 0,Y 133.427,Z 593.614,A -85,B 0,C 180,E1 -27202.145,E2 -27202.145} C_VEL
LIN {X 0,Y 136.673,Z 588.869,A -85,B 0,C 180,E1 -27204.696,E2 -27204.696} C_VEL
LIN {X 0,Y 140.654,Z 581.977,A -85,B 0,C 180,E1 -27207.267,E2 -27207.267} C_VEL
LIN {X 0,Y 144.459,Z 574.355,A -85,B 0,C 180,E1 -27209.311,E2 -27209.311} C_VEL
LIN {X 0,Y 141.627,Z 603.627,A -85,B 0,C 180,E1 -27210.422,E2 -27210.422} C_VEL
LIN {X 0,Y 138.923,Z 617.135,A -85,B 0,C 180,E1 -27211.21,E2 -27211.21} C_VEL
LIN {X 0,Y 135.311,Z 629.879,A -85,B 0,C 180,E1 -27212.433,E2 -27212.433} C_VEL
LIN {X 0,Y 131.252,Z 640.739,A -85,B 0,C 180,E1 -27213.906,E2 -27213.906} C_VEL
LIN {X 0,Y 125.935,Z 652.05,A -85,B 0,C 180,E1 -27215.983,E2 -27215.983} C_VEL
LIN {X 0,Y 120.203,Z 662.252,A -85,B 0,C 180,E1 -27218.556,E2 -27218.556} C_VEL
LIN {X 0,Y 114.689,Z 670.612,A -85,B 0,C 180,E1 -27221.353,E2 -27221.353} C_VEL
LIN {X 0,Y 108.005,Z 679.598,A -85,B 0,C 180,E1 -27225.549,E2 -27225.549} C_VEL
LIN {X 0,Y 101.794,Z 686.92,A -85,B 0,C 180,E1 -27230.31,E2 -27230.31} C_VEL
LIN {X 0,Y 97.225,Z 691.838,A -85,B 0,C 180,E1 -27234.67,E2 -27234.67} C_VEL
LIN {X 0,Y 92.404,Z 696.594,A -85,B 0,C 180,E1 -27240.372,E2 -27240.372} C_VEL
LIN {X 0,Y 88.709,Z 700.23,A -85,B 0,C 180,E1 -27246.664,E2 -27246.664} C_VEL
LIN {X 0,Y 86.773,Z 702.101,A -85,B 0,C 180,E1 -27251.097,E2 -27251.097} C_VEL
LIN {X 0,Y 85.342,Z 703.524,A -85,B 0,C 180,E1 -27255.697,E2 -27255.697} C_VEL
LIN {X 0,Y 84.388,Z 704.522,A -85,B 0,C 180,E1 -27260.412,E2 -27260.412} C_VEL
LIN {X 0,Y 83.887,Z 705.135,A -85,B 0,C 180,E1 -27265.195,E2 -27265.195} C_VEL
LIN {X 0,Y 83.817,Z 705.364,A -85,B 0,C 180,E1 -27270.001,E2 -27270.001} C_VEL
LIN {X 0,Y 83.884,Z 705.162,A -85,B 0,C 180,E1 -27274.807,E2 -27274.807} C_VEL
LIN {X 0,Y 84.361,Z 704.566,A -85,B 0,C 180,E1 -27279.592,E2 -27279.592} C_VEL
LIN {X 0,Y 85.274,Z 703.586,A -85,B 0,C 180,E1 -27284.316,E2 -27284.316} C_VEL
LIN {X 0,Y 86.716,Z 702.199,A -85,B 0,C 180,E1 -27288.917,E2 -27288.917} C_VEL
LIN {X 0,Y 89.735,Z 699.29,A -85,B 0,C 180,E1 -27295.516,E2 -27295.516} C_VEL
LIN {X 0,Y 93.858,Z 695.337,A -85,B 0,C 180,E1 -27301.612,E2 -27301.612} C_VEL
LIN {X 0,Y 98.947,Z 690.212,A -85,B 0,C 180,E1 -27307.139,E2 -27307.139} C_VEL
LIN {X 0,Y 105.633,Z 682.791,A -85,B 0,C 180,E1 -27312.73,E2 -27312.73} C_VEL
LIN {X 0,Y 111.156,Z 675.729,A -85,B 0,C 180,E1 -27316.645,E2 -27316.645} C_VEL
LIN {X 0,Y 116.999,Z 667.513,A -85,B 0,C 180,E1 -27319.986,E2 -27319.986} C_VEL
LIN {X 0,Y 123.29,Z 657.367,A -85,B 0,C 180,E1 -27322.946,E2 -27322.946} C_VEL
LIN {X 0,Y 129.164,Z 645.953,A -85,B 0,C 180,E1 -27325.385,E2 -27325.385} C_VEL
LIN {X 0,Y 133.856,Z 634.628,A -85,B 0,C 180,E1 -27327.149,E2 -27327.149} C_VEL
LIN {X 0,Y 138.001,Z 621.734,A -85,B 0,C 180,E1 -27328.544,E2 -27328.544} C_VEL
LIN {X 0,Y 140.923,Z 609.085,A -85,B 0,C 180,E1 -27329.47,E2 -27329.47} C_VEL
LIN {X 0,Y 142.847,Z 595.031,A -85,B 0,C 180,E1 -27330.085,E2 -27330.085} C_VEL
LIN {X 0,Y 147.332,Z 545.911,A -85,B 0,C 180,E1 -27331.802,E2 -27331.802} C_VEL
LIN {X 0,Y 147.309,Z 534.776,A -85,B 0,C 180,E1 -27332.964,E2 -27332.964} C_VEL
LIN {X 0,Y 144.246,Z 526.036,A -85,B 0,C 180,E1 -27336.489,E2 -27336.489} C_VEL
LIN {X 0,Y 141.807,Z 520.025,A -85,B 0,C 180,E1 -27339.701,E2 -27339.701} C_VEL
LIN {X 0,Y 139.349,Z 514.474,A -85,B 0,C 180,E1 -27343.584,E2 -27343.584} C_VEL
LIN {X 0,Y 136.805,Z 509.134,A -85,B 0,C 180,E1 -27349.033,E2 -27349.033} C_VEL
LIN {X 0,Y 135.469,Z 506.272,A -85,B 0,C 180,E1 -27353.671,E2 -27353.671} C_VEL
LIN {X 0,Y 134.909,Z 503.925,A -85,B 0,C 180,E1 -27360,E2 -27360} C_VEL
LIN {X 0,Y 135.146,Z 503.993,A -85,B 0,C 180,E1 -27363.54,E2 -27363.54} C_VEL
LIN {X 0,Y 136.655,Z 506.307,A -85,B 0,C 180,E1 -27369.996,E2 -27369.996} C_VEL
LIN {X 0,Y 138.84,Z 509.227,A -85,B 0,C 180,E1 -27374.848,E2 -27374.848} C_VEL
LIN {X 0,Y 142.356,Z 514.76,A -85,B 0,C 180,E1 -27380.312,E2 -27380.312} C_VEL
LIN {X 0,Y 145.928,Z 521.158,A -85,B 0,C 180,E1 -27384.582,E2 -27384.582} C_VEL
LIN {X 0,Y 147.44,Z 524.106,A -85,B 0,C 180,E1 -27386.163,E2 -27386.163} C_VEL
LIN {X 0,Y 146.963,Z 547.214,A -85,B 0,C 180,E1 -27388.221,E2 -27388.221} C_VEL
LIN {X 0,Y 141.667,Z 603.693,A -85,B 0,C 180,E1 -27390.243,E2 -27390.243} C_VEL
LIN {X 0,Y 139.314,Z 616.409,A -85,B 0,C 180,E1 -27390.95,E2 -27390.95} C_VEL
LIN {X 0,Y 135.759,Z 629.142,A -85,B 0,C 180,E1 -27392.036,E2 -27392.036} C_VEL
LIN {X 0,Y 131.651,Z 640.492,A -85,B 0,C 180,E1 -27393.475,E2 -27393.475} C_VEL
LIN {X 0,Y 126.323,Z 652.163,A -85,B 0,C 180,E1 -27395.544,E2 -27395.544} C_VEL
LIN {X 0,Y 120.498,Z 662.583,A -85,B 0,C 180,E1 -27398.057,E2 -27398.057} C_VEL
LIN {X 0,Y 114.339,Z 671.981,A -85,B 0,C 180,E1 -27401.151,E2 -27401.151} C_VEL
LIN {X 0,Y 107.478,Z 681.002,A -85,B 0,C 180,E1 -27405.335,E2 -27405.335} C_VEL
LIN {X 0,Y 101.517,Z 688.18,A -85,B 0,C 180,E1 -27410.085,E2 -27410.085} C_VEL
LIN {X 0,Y 96.766,Z 693.173,A -85,B 0,C 180,E1 -27414.476,E2 -27414.476} C_VEL
LIN {X 0,Y 92.049,Z 697.926,A -85,B 0,C 180,E1 -27420.245,E2 -27420.245} C_VEL
LIN {X 0,Y 88.312,Z 701.553,A -85,B 0,C 180,E1 -27426.552,E2 -27426.552} C_VEL
LIN {X 0,Y 86.488,Z 703.423,A -85,B 0,C 180,E1 -27431.031,E2 -27431.031} C_VEL
LIN {X 0,Y 85.128,Z 704.829,A -85,B 0,C 180,E1 -27435.659,E2 -27435.659} C_VEL
LIN {X 0,Y 84.292,Z 705.824,A -85,B 0,C 180,E1 -27440.4,E2 -27440.4} C_VEL
LIN {X 0,Y 83.877,Z 706.431,A -85,B 0,C 180,E1 -27445.193,E2 -27445.193} C_VEL
LIN {X 0,Y 83.885,Z 706.642,A -85,B 0,C 180,E1 -27449.999,E2 -27449.999} C_VEL
LIN {X 0,Y 83.877,Z 706.413,A -85,B 0,C 180,E1 -27454.806,E2 -27454.806} C_VEL
LIN {X 0,Y 84.292,Z 705.795,A -85,B 0,C 180,E1 -27459.599,E2 -27459.599} C_VEL
LIN {X 0,Y 85.128,Z 704.788,A -85,B 0,C 180,E1 -27464.339,E2 -27464.339} C_VEL
LIN {X 0,Y 86.489,Z 703.358,A -85,B 0,C 180,E1 -27468.967,E2 -27468.967} C_VEL
LIN {X 0,Y 89.417,Z 700.394,A -85,B 0,C 180,E1 -27475.612,E2 -27475.612} C_VEL
LIN {X 0,Y 93.543,Z 696.375,A -85,B 0,C 180,E1 -27481.73,E2 -27481.73} C_VEL
LIN {X 0,Y 98.562,Z 691.181,A -85,B 0,C 180,E1 -27487.307,E2 -27487.307} C_VEL
LIN {X 0,Y 104.367,Z 684.646,A -85,B 0,C 180,E1 -27492.329,E2 -27492.329} C_VEL
LIN {X 0,Y 110.812,Z 676.515,A -85,B 0,C 180,E1 -27496.832,E2 -27496.832} C_VEL
LIN {X 0,Y 116.756,Z 668.171,A -85,B 0,C 180,E1 -27500.127,E2 -27500.127} C_VEL
LIN {X 0,Y 122.076,Z 659.565,A -85,B 0,C 180,E1 -27502.68,E2 -27502.68} C_VEL
LIN {X 0,Y 122.464,Z 657.983,A -85,B 0,C 180,E1 -27503.395,E2 -27503.395} C_VEL
LIN {X 0,Y 122.005,Z 656.901,A -85,B 0,C 180,E1 -27504.351,E2 -27504.351} C_VEL
LIN {X 0,Y 120.06,Z 655.995,A -85,B 0,C 180,E1 -27506.24,E2 -27506.24} C_VEL
LIN {X 0,Y 113.905,Z 655.846,A -85,B 0,C 180,E1 -27511.213,E2 -27511.213} C_VEL
LIN {X 0,Y 113.289,Z 655.625,A -85,B 0,C 180,E1 -27511.946,E2 -27511.946} C_VEL
LIN {X 0,Y 108.107,Z 652.297,A -85,B 0,C 180,E1 -27521.032,E2 -27521.032} C_VEL
LIN {X 0,Y 106.926,Z 649.512,A -85,B 0,C 180,E1 -27526.7,E2 -27526.7} C_VEL
LIN {X 0,Y 107.463,Z 645.481,A -85,B 0,C 180,E1 -27532.484,E2 -27532.484} C_VEL
LIN {X 0,Y 111.19,Z 636.905,A -85,B 0,C 180,E1 -27541.811,E2 -27541.811} C_VEL
LIN {X 0,Y 114.016,Z 632.563,A -85,B 0,C 180,E1 -27547.082,E2 -27547.082} C_VEL
LIN {X 0,Y 117.508,Z 627.502,A -85,B 0,C 180,E1 -27551.209,E2 -27551.209} C_VEL
LIN {X 0,Y 122.332,Z 620.451,A -85,B 0,C 180,E1 -27555.575,E2 -27555.575} C_VEL
LIN {X 0,Y 128.103,Z 611.132,A -85,B 0,C 180,E1 -27559.844,E2 -27559.844} C_VEL
LIN {X 0,Y 134.578,Z 599.073,A -85,B 0,C 180,E1 -27564.079,E2 -27564.079} C_VEL
LIN {X 0,Y 138.195,Z 594.035,A -85,B 0,C 180,E1 -27566.626,E2 -27566.626} C_VEL
LIN {X 0,Y 139.4,Z 592.153,A -85,B 0,C 180,E1 -27567.39,E2 -27567.39} C_VEL
LIN {X 0,Y 137.563,Z 607.227,A -85,B 0,C 180,E1 -27568.065,E2 -27568.065} C_VEL
LIN {X 0,Y 134.834,Z 619.33,A -85,B 0,C 180,E1 -27568.798,E2 -27568.798} C_VEL
LIN {X 0,Y 130.947,Z 631.885,A -85,B 0,C 180,E1 -27570.068,E2 -27570.068} C_VEL
LIN {X 0,Y 126.741,Z 642.322,A -85,B 0,C 180,E1 -27571.508,E2 -27571.508} C_VEL
LIN {X 0,Y 121.22,Z 653.358,A -85,B 0,C 180,E1 -27573.548,E2 -27573.548} C_VEL
LIN {X 0,Y 115.268,Z 663.327,A -85,B 0,C 180,E1 -27576.112,E2 -27576.112} C_VEL
LIN {X 0,Y 108.876,Z 672.306,A -85,B 0,C 180,E1 -27579.231,E2 -27579.231} C_VEL
LIN {X 0,Y 101.563,Z 681.407,A -85,B 0,C 180,E1 -27583.788,E2 -27583.788} C_VEL
LIN {X 0,Y 95.384,Z 688.057,A -85,B 0,C 180,E1 -27588.461,E2 -27588.461} C_VEL
LIN {X 0,Y 89.665,Z 693.623,A -85,B 0,C 180,E1 -27593.996,E2 -27593.996} C_VEL
LIN {X 0,Y 84.769,Z 697.989,A -85,B 0,C 180,E1 -27600.17,E2 -27600.17} C_VEL
LIN {X 0,Y 82.215,Z 700.284,A -85,B 0,C 180,E1 -27604.697,E2 -27604.697} C_VEL
LIN {X 0,Y 80.082,Z 702.156,A -85,B 0,C 180,E1 -27609.45,E2 -27609.45} C_VEL
LIN {X 0,Y 78.474,Z 703.578,A -85,B 0,C 180,E1 -27614.415,E2 -27614.415} C_VEL
LIN {X 0,Y 77.391,Z 704.576,A -85,B 0,C 180,E1 -27619.536,E2 -27619.536} C_VEL
LIN {X 0,Y 76.811,Z 705.189,A -85,B 0,C 180,E1 -27624.751,E2 -27624.751} C_VEL
LIN {X 0,Y 76.739,Z 705.418,A -85,B 0,C 180,E1 -27630.001,E2 -27630.001} C_VEL
LIN {X 0,Y 76.808,Z 705.216,A -85,B 0,C 180,E1 -27635.251,E2 -27635.251} C_VEL
LIN {X 0,Y 77.365,Z 704.62,A -85,B 0,C 180,E1 -27640.469,E2 -27640.469} C_VEL
LIN {X 0,Y 78.416,Z 703.639,A -85,B 0,C 180,E1 -27645.598,E2 -27645.598} C_VEL
LIN {X 0,Y 80.031,Z 702.252,A -85,B 0,C 180,E1 -27650.565,E2 -27650.565} C_VEL
LIN {X 0,Y 83.365,Z 699.343,A -85,B 0,C 180,E1 -27657.625,E2 -27657.625} C_VEL
LIN {X 0,Y 87.868,Z 695.388,A -85,B 0,C 180,E1 -27664.049,E2 -27664.049} C_VEL
LIN {X 0,Y 93.356,Z 690.263,A -85,B 0,C 180,E1 -27669.785,E2 -27669.785} C_VEL
LIN {X 0,Y 99.64,Z 683.803,A -85,B 0,C 180,E1 -27674.858,E2 -27674.858} C_VEL
LIN {X 0,Y 106.4,Z 675.776,A -85,B 0,C 180,E1 -27679.43,E2 -27679.43} C_VEL
LIN {X 0,Y 112.572,Z 667.558,A -85,B 0,C 180,E1 -27682.751,E2 -27682.751} C_VEL
LIN {X 0,Y 119.146,Z 657.409,A -85,B 0,C 180,E1 -27685.672,E2 -27685.672} C_VEL
LIN {X 0,Y 125.273,Z 645.989,A -85,B 0,C 180,E1 -27688.054,E2 -27688.054} C_VEL
LIN {X 0,Y 130.148,Z 634.655,A -85,B 0,C 180,E1 -27689.77,E2 -27689.77} C_VEL
LIN {X 0,Y 134.441,Z 621.75,A -85,B 0,C 180,E1 -27691.12,E2 -27691.12} C_VEL
LIN {X 0,Y 137.479,Z 608.919,A -85,B 0,C 180,E1 -27692.03,E2 -27692.03} C_VEL
LIN {X 0,Y 139.476,Z 594.67,A -85,B 0,C 180,E1 -27692.618,E2 -27692.618} C_VEL
LIN {X 0,Y 144.034,Z 546.421,A -85,B 0,C 180,E1 -27694.29,E2 -27694.29} C_VEL
LIN {X 0,Y 144.06,Z 538.149,A -85,B 0,C 180,E1 -27695.212,E2 -27695.212} C_VEL
LIN {X 0,Y 141.369,Z 530.092,A -85,B 0,C 180,E1 -27698.759,E2 -27698.759} C_VEL
LIN {X 0,Y 139.156,Z 524.242,A -85,B 0,C 180,E1 -27702.17,E2 -27702.17} C_VEL
LIN {X 0,Y 137.055,Z 519.21,A -85,B 0,C 180,E1 -27706.163,E2 -27706.163} C_VEL
LIN {X 0,Y 135.128,Z 514.748,A -85,B 0,C 180,E1 -27711.4,E2 -27711.4} C_VEL
LIN {X 0,Y 134.112,Z 512.009,A -85,B 0,C 180,E1 -27716.996,E2 -27716.996} C_VEL
LIN {X 0,Y 134.041,Z 511.002,A -85,B 0,C 180,E1 -27720,E2 -27720} C_VEL
LIN {X 0,Y 134.276,Z 511.097,A -85,B 0,C 180,E1 -27723.563,E2 -27723.563} C_VEL
LIN {X 0,Y 135.787,Z 513.495,A -85,B 0,C 180,E1 -27730.06,E2 -27730.06} C_VEL
LIN {X 0,Y 137.766,Z 516.401,A -85,B 0,C 180,E1 -27734.587,E2 -27734.587} C_VEL
LIN {X 0,Y 140.803,Z 521.51,A -85,B 0,C 180,E1 -27739.557,E2 -27739.557} C_VEL
LIN {X 0,Y 144.024,Z 527.693,A -85,B 0,C 180,E1 -27743.672,E2 -27743.672} C_VEL
LIN {X 0,Y 144.29,Z 528.341,A -85,B 0,C 180,E1 -27743.991,E2 -27743.991} C_VEL
LIN {X 0,Y 143.617,Z 548.819,A -85,B 0,C 180,E1 -27745.794,E2 -27745.794} C_VEL
LIN {X 0,Y 138.144,Z 604.373,A -85,B 0,C 180,E1 -27747.727,E2 -27747.727} C_VEL
LIN {X 0,Y 135.619,Z 617.134,A -85,B 0,C 180,E1 -27748.435,E2 -27748.435} C_VEL
LIN {X 0,Y 131.783,Z 630.214,A -85,B 0,C 180,E1 -27749.546,E2 -27749.546} C_VEL
LIN {X 0,Y 127.165,Z 642.088,A -85,B 0,C 180,E1 -27751.058,E2 -27751.058} C_VEL
LIN {X 0,Y 121.655,Z 653.392,A -85,B 0,C 180,E1 -27753.105,E2 -27753.105} C_VEL
LIN {X 0,Y 115.584,Z 663.593,A -85,B 0,C 180,E1 -27755.583,E2 -27755.583} C_VEL
LIN {X 0,Y 109.801,Z 671.935,A -85,B 0,C 180,E1 -27758.363,E2 -27758.363} C_VEL
LIN {X 0,Y 102.54,Z 680.954,A -85,B 0,C 180,E1 -27762.54,E2 -27762.54} C_VEL
LIN {X 0,Y 96.77,Z 687.434,A -85,B 0,C 180,E1 -27766.8,E2 -27766.8} C_VEL
LIN {X 0,Y 91.063,Z 693.122,A -85,B 0,C 180,E1 -27771.871,E2 -27771.871} C_VEL
LIN {X 0,Y 85.941,Z 697.874,A -85,B 0,C 180,E1 -27777.889,E2 -27777.889} C_VEL
LIN {X 0,Y 81.81,Z 701.5,A -85,B 0,C 180,E1 -27784.561,E2 -27784.561} C_VEL
LIN {X 0,Y 79.774,Z 703.37,A -85,B 0,C 180,E1 -27789.365,E2 -27789.365} C_VEL
LIN {X 0,Y 78.249,Z 704.776,A -85,B 0,C 180,E1 -27794.368,E2 -27794.368} C_VEL
LIN {X 0,Y 77.283,Z 705.77,A -85,B 0,C 180,E1 -27799.52,E2 -27799.52} C_VEL
LIN {X 0,Y 76.799,Z 706.377,A -85,B 0,C 180,E1 -27804.749,E2 -27804.749} C_VEL
LIN {X 0,Y 76.784,Z 706.588,A -85,B 0,C 180,E1 -27809.999,E2 -27809.999} C_VEL
LIN {X 0,Y 76.799,Z 706.359,A -85,B 0,C 180,E1 -27815.25,E2 -27815.25} C_VEL
LIN {X 0,Y 77.283,Z 705.74,A -85,B 0,C 180,E1 -27820.478,E2 -27820.478} C_VEL
LIN {X 0,Y 78.249,Z 704.734,A -85,B 0,C 180,E1 -27825.631,E2 -27825.631} C_VEL
LIN {X 0,Y 79.776,Z 703.303,A -85,B 0,C 180,E1 -27830.633,E2 -27830.633} C_VEL
LIN {X 0,Y 83.056,Z 700.34,A -85,B 0,C 180,E1 -27837.735,E2 -27837.735} C_VEL
LIN {X 0,Y 87.577,Z 696.321,A -85,B 0,C 180,E1 -27844.176,E2 -27844.176} C_VEL
LIN {X 0,Y 93.013,Z 691.127,A -85,B 0,C 180,E1 -27849.96,E2 -27849.96} C_VEL
LIN {X 0,Y 99.21,Z 684.592,A -85,B 0,C 180,E1 -27855.104,E2 -27855.104} C_VEL
LIN {X 0,Y 106.066,Z 676.463,A -85,B 0,C 180,E1 -27859.64,E2 -27859.64} C_VEL
LIN {X 0,Y 112.324,Z 668.121,A -85,B 0,C 180,E1 -27862.916,E2 -27862.916} C_VEL
LIN {X 0,Y 118.238,Z 658.964,A -85,B 0,C 180,E1 -27865.56,E2 -27865.56} C_VEL
LIN {X 0,Y 118.221,Z 657.802,A -85,B 0,C 180,E1 -27866.333,E2 -27866.333} C_VEL
LIN {X 0,Y 113.289,Z 655.625,A -85,B 0,C 180,E1 -27871.946,E2 -27871.946} C_VEL
LIN {X 0,Y 111.539,Z 655.494,A -85,B 0,C 180,E1 -27873.785,E2 -27873.785} C_VEL
LIN {X 0,Y 104.612,Z 657.855,A -85,B 0,C 180,E1 -27879.833,E2 -27879.833} C_VEL
LIN {X 0,Y 103.523,Z 657.547,A -85,B 0,C 180,E1 -27881.921,E2 -27881.921} C_VEL
LIN {X 0,Y 102.81,Z 653.788,A -85,B 0,C 180,E1 -27889.61,E2 -27889.61} C_VEL
LIN {X 0,Y 104.467,Z 649.126,A -85,B 0,C 180,E1 -27896.143,E2 -27896.143} C_VEL
LIN {X 0,Y 108.44,Z 642.411,A -85,B 0,C 180,E1 -27903.716,E2 -27903.716} C_VEL
LIN {X 0,Y 111.864,Z 638.109,A -85,B 0,C 180,E1 -27909.037,E2 -27909.037} C_VEL
LIN {X 0,Y 115.774,Z 633.301,A -85,B 0,C 180,E1 -27913.062,E2 -27913.062} C_VEL
LIN {X 0,Y 121.777,Z 625.717,A -85,B 0,C 180,E1 -27917.783,E2 -27917.783} C_VEL
LIN {X 0,Y 128.426,Z 616.36,A -85,B 0,C 180,E1 -27921.995,E2 -27921.995} C_VEL
LIN {X 0,Y 134.442,Z 606.545,A -85,B 0,C 180,E1 -27925.315,E2 -27925.315} C_VEL
LIN {X 0,Y 131.711,Z 618.816,A -85,B 0,C 180,E1 -27926.058,E2 -27926.058} C_VEL
LIN {X 0,Y 127.849,Z 631.091,A -85,B 0,C 180,E1 -27927.204,E2 -27927.204} C_VEL
LIN {X 0,Y 123.179,Z 642.366,A -85,B 0,C 180,E1 -27928.691,E2 -27928.691} C_VEL
LIN {X 0,Y 117.454,Z 653.405,A -85,B 0,C 180,E1 -27930.668,E2 -27930.668} C_VEL
LIN {X 0,Y 111.226,Z 663.377,A -85,B 0,C 180,E1 -27933.153,E2 -27933.153} C_VEL
LIN {X 0,Y 104.528,Z 672.357,A -85,B 0,C 180,E1 -27936.213,E2 -27936.213} C_VEL
LIN {X 0,Y 97.311,Z 680.85,A -85,B 0,C 180,E1 -27940.383,E2 -27940.383} C_VEL
LIN {X 0,Y 91.326,Z 687.027,A -85,B 0,C 180,E1 -27944.616,E2 -27944.616} C_VEL
LIN {X 0,Y 84.016,Z 693.677,A -85,B 0,C 180,E1 -27951.143,E2 -27951.143} C_VEL
LIN {X 0,Y 78.668,Z 698.043,A -85,B 0,C 180,E1 -27957.587,E2 -27957.587} C_VEL
LIN {X 0,Y 75.84,Z 700.339,A -85,B 0,C 180,E1 -27962.398,E2 -27962.398} C_VEL
LIN {X 0,Y 73.475,Z 702.21,A -85,B 0,C 180,E1 -27967.506,E2 -27967.506} C_VEL
LIN {X 0,Y 71.663,Z 703.632,A -85,B 0,C 180,E1 -27972.891,E2 -27972.891} C_VEL
LIN {X 0,Y 69.758,Z 705.244,A -85,B 0,C 180,E1 -27984.218,E2 -27984.218} C_VEL
LIN {X 0,Y 69.652,Z 705.472,A -85,B 0,C 180,E1 -27990.001,E2 -27990.001} C_VEL
LIN {X 0,Y 69.754,Z 705.27,A -85,B 0,C 180,E1 -27995.783,E2 -27995.783} C_VEL
LIN {X 0,Y 70.385,Z 704.674,A -85,B 0,C 180,E1 -28001.52,E2 -28001.52} C_VEL
LIN {X 0,Y 71.582,Z 703.693,A -85,B 0,C 180,E1 -28007.131,E2 -28007.131} C_VEL
LIN {X 0,Y 73.413,Z 702.305,A -85,B 0,C 180,E1 -28012.516,E2 -28012.516} C_VEL
LIN {X 0,Y 77.11,Z 699.395,A -85,B 0,C 180,E1 -28020.086,E2 -28020.086} C_VEL
LIN {X 0,Y 82.066,Z 695.44,A -85,B 0,C 180,E1 -28026.833,E2 -28026.833} C_VEL
LIN {X 0,Y 87.994,Z 690.313,A -85,B 0,C 180,E1 -28032.758,E2 -28032.758} C_VEL
LIN {X 0,Y 94.725,Z 683.853,A -85,B 0,C 180,E1 -28037.898,E2 -28037.898} C_VEL
LIN {X 0,Y 101.914,Z 675.824,A -85,B 0,C 180,E1 -28042.472,E2 -28042.472} C_VEL
LIN {X 0,Y 108.431,Z 667.603,A -85,B 0,C 180,E1 -28045.732,E2 -28045.732} C_VEL
LIN {X 0,Y 115.292,Z 657.45,A -85,B 0,C 180,E1 -28048.587,E2 -28048.587} C_VEL
LIN {X 0,Y 121.671,Z 646.025,A -85,B 0,C 180,E1 -28050.888,E2 -28050.888} C_VEL
LIN {X 0,Y 126.72,Z 634.683,A -85,B 0,C 180,E1 -28052.546,E2 -28052.546} C_VEL
LIN {X 0,Y 131.168,Z 621.765,A -85,B 0,C 180,E1 -28053.829,E2 -28053.829} C_VEL
LIN {X 0,Y 134.31,Z 608.868,A -85,B 0,C 180,E1 -28054.701,E2 -28054.701} C_VEL
LIN {X 0,Y 136.4,Z 594.238,A -85,B 0,C 180,E1 -28055.273,E2 -28055.273} C_VEL
LIN {X 0,Y 141.002,Z 547.207,A -85,B 0,C 180,E1 -28056.871,E2 -28056.871} C_VEL
LIN {X 0,Y 141.104,Z 541.964,A -85,B 0,C 180,E1 -28057.444,E2 -28057.444} C_VEL
LIN {X 0,Y 138.913,Z 534.739,A -85,B 0,C 180,E1 -28060.801,E2 -28060.801} C_VEL
LIN {X 0,Y 137.063,Z 529.525,A -85,B 0,C 180,E1 -28064.096,E2 -28064.096} C_VEL
LIN {X 0,Y 135.612,Z 525.655,A -85,B 0,C 180,E1 -28067.276,E2 -28067.276} C_VEL
LIN {X 0,Y 134.068,Z 521.627,A -85,B 0,C 180,E1 -28071.996,E2 -28071.996} C_VEL
LIN {X 0,Y 133.215,Z 519.044,A -85,B 0,C 180,E1 -28077.259,E2 -28077.259} C_VEL
LIN {X 0,Y 133.167,Z 518.13,A -85,B 0,C 180,E1 -28080,E2 -28080} C_VEL
LIN {X 0,Y 133.412,Z 518.16,A -85,B 0,C 180,E1 -28083.586,E2 -28083.586} C_VEL
LIN {X 0,Y 134.724,Z 520.446,A -85,B 0,C 180,E1 -28089.571,E2 -28089.571} C_VEL
LIN {X 0,Y 136.351,Z 522.947,A -85,B 0,C 180,E1 -28093.601,E2 -28093.601} C_VEL
LIN {X 0,Y 139.035,Z 527.8,A -85,B 0,C 180,E1 -28098.417,E2 -28098.417} C_VEL
LIN {X 0,Y 141.34,Z 532.539,A -85,B 0,C 180,E1 -28101.705,E2 -28101.705} C_VEL
LIN {X 0,Y 140.555,Z 550.174,A -85,B 0,C 180,E1 -28103.238,E2 -28103.238} C_VEL
LIN {X 0,Y 135.043,Z 604.078,A -85,B 0,C 180,E1 -28105.053,E2 -28105.053} C_VEL
LIN {X 0,Y 132.389,Z 617.125,A -85,B 0,C 180,E1 -28105.735,E2 -28105.735} C_VEL
LIN {X 0,Y 128.431,Z 630.191,A -85,B 0,C 180,E1 -28106.79,E2 -28106.79} C_VEL
LIN {X 0,Y 123.662,Z 642.054,A -85,B 0,C 180,E1 -28108.247,E2 -28108.247} C_VEL
LIN {X 0,Y 117.929,Z 653.353,A -85,B 0,C 180,E1 -28110.215,E2 -28110.215} C_VEL
LIN {X 0,Y 111.601,Z 663.549,A -85,B 0,C 180,E1 -28112.617,E2 -28112.617} C_VEL
LIN {X 0,Y 105.543,Z 671.889,A -85,B 0,C 180,E1 -28115.341,E2 -28115.341} C_VEL
LIN {X 0,Y 97.859,Z 680.905,A -85,B 0,C 180,E1 -28119.461,E2 -28119.461} C_VEL
LIN {X 0,Y 91.223,Z 687.865,A -85,B 0,C 180,E1 -28124.127,E2 -28124.127} C_VEL
LIN {X 0,Y 85.581,Z 693.071,A -85,B 0,C 180,E1 -28128.93,E2 -28128.93} C_VEL
LIN {X 0,Y 79.994,Z 697.822,A -85,B 0,C 180,E1 -28135.174,E2 -28135.174} C_VEL
LIN {X 0,Y 75.427,Z 701.447,A -85,B 0,C 180,E1 -28142.232,E2 -28142.232} C_VEL
LIN {X 0,Y 73.148,Z 703.317,A -85,B 0,C 180,E1 -28147.398,E2 -28147.398} C_VEL
LIN {X 0,Y 71.427,Z 704.722,A -85,B 0,C 180,E1 -28152.83,E2 -28152.83} C_VEL
LIN {X 0,Y 70.309,Z 705.717,A -85,B 0,C 180,E1 -28158.467,E2 -28158.467} C_VEL
LIN {X 0,Y 69.743,Z 706.323,A -85,B 0,C 180,E1 -28164.216,E2 -28164.216} C_VEL
LIN {X 0,Y 69.705,Z 706.534,A -85,B 0,C 180,E1 -28169.999,E2 -28169.999} C_VEL
LIN {X 0,Y 69.743,Z 706.304,A -85,B 0,C 180,E1 -28175.783,E2 -28175.783} C_VEL
LIN {X 0,Y 70.309,Z 705.686,A -85,B 0,C 180,E1 -28181.531,E2 -28181.531} C_VEL
LIN {X 0,Y 71.427,Z 704.679,A -85,B 0,C 180,E1 -28187.168,E2 -28187.168} C_VEL
LIN {X 0,Y 73.149,Z 703.248,A -85,B 0,C 180,E1 -28192.6,E2 -28192.6} C_VEL
LIN {X 0,Y 76.835,Z 700.285,A -85,B 0,C 180,E1 -28200.203,E2 -28200.203} C_VEL
LIN {X 0,Y 81.795,Z 696.267,A -85,B 0,C 180,E1 -28206.974,E2 -28206.974} C_VEL
LIN {X 0,Y 87.689,Z 691.073,A -85,B 0,C 180,E1 -28212.941,E2 -28212.941} C_VEL
LIN {X 0,Y 94.317,Z 684.539,A -85,B 0,C 180,E1 -28218.171,E2 -28218.171} C_VEL
LIN {X 0,Y 101.612,Z 676.411,A -85,B 0,C 180,E1 -28222.693,E2 -28222.693} C_VEL
LIN {X 0,Y 108.184,Z 668.07,A -85,B 0,C 180,E1 -28225.922,E2 -28225.922} C_VEL
LIN {X 0,Y 111.122,Z 663.881,A -85,B 0,C 180,E1 -28227.218,E2 -28227.218} C_VEL
LIN {X 0,Y 111.296,Z 662.234,A -85,B 0,C 180,E1 -28228.399,E2 -28228.399} C_VEL
LIN {X 0,Y 103.523,Z 657.547,A -85,B 0,C 180,E1 -28241.921,E2 -28241.921} C_VEL
LIN {X 0,Y 102.646,Z 657.118,A -85,B 0,C 180,E1 -28244.099,E2 -28244.099} C_VEL
LIN {X 0,Y 99.065,Z 657.998,A -85,B 0,C 180,E1 -28251.498,E2 -28251.498} C_VEL
LIN {X 0,Y 99.161,Z 657.199,A -85,B 0,C 180,E1 -28253.724,E2 -28253.724} C_VEL
LIN {X 0,Y 103.093,Z 650.896,A -85,B 0,C 180,E1 -28261.954,E2 -28261.954} C_VEL
LIN {X 0,Y 106.136,Z 647.114,A -85,B 0,C 180,E1 -28266.662,E2 -28266.662} C_VEL
LIN {X 0,Y 109.575,Z 643.528,A -85,B 0,C 180,E1 -28271.094,E2 -28271.094} C_VEL
LIN {X 0,Y 114.096,Z 638.739,A -85,B 0,C 180,E1 -28275.176,E2 -28275.176} C_VEL
LIN {X 0,Y 121.594,Z 630.414,A -85,B 0,C 180,E1 -28280.292,E2 -28280.292} C_VEL
LIN {X 0,Y 127.001,Z 623.766,A -85,B 0,C 180,E1 -28283.299,E2 -28283.299} C_VEL
LIN {X 0,Y 126.953,Z 624.879,A -85,B 0,C 180,E1 -28283.696,E2 -28283.696} C_VEL
LIN {X 0,Y 122.151,Z 637.489,A -85,B 0,C 180,E1 -28285.018,E2 -28285.018} C_VEL
LIN {X 0,Y 116.205,Z 649.638,A -85,B 0,C 180,E1 -28286.866,E2 -28286.866} C_VEL
LIN {X 0,Y 109.635,Z 660.307,A -85,B 0,C 180,E1 -28289.142,E2 -28289.142} C_VEL
